   //    movement227ExecutabilityRight : Bool;   // Setup screen: executability of movement right
   //    movement228ExecutabilityLeft : Bool;   // Setup screen: executability of movement left
   //    movement228ExecutabilityRight : Bool;   // Setup screen: executability of movement right
   //    movement229ExecutabilityLeft : Bool;   // Setup screen: executability of movement left
   //    movement229ExecutabilityRight : Bool;   // Setup screen: executability of movement right
   //    movement230ExecutabilityLeft : Bool;   // Setup screen: executability of movement left
   //    movement230ExecutabilityRight : Bool;   // Setup screen: executability of movement right
   //    movement231ExecutabilityLeft : Bool;   // Setup screen: executability of movement left
   //    movement231ExecutabilityRight : Bool;   // Setup screen: executability of movement right
   //    movement232ExecutabilityLeft : Bool;   // Setup screen: executability of movement left
   //    movement232ExecutabilityRight : Bool;   // Setup screen: executability of movement right
   //    movement233ExecutabilityLeft : Bool;   // Setup screen: executability of movement left
   //    movement233ExecutabilityRight : Bool;   // Setup screen: executability of movement right
   //    movement234ExecutabilityLeft : Bool;   // Setup screen: executability of movement left
   //    movement234ExecutabilityRight : Bool;   // Setup screen: executability of movement right
   //    movement235ExecutabilityLeft : Bool;   // Setup screen: executability of movement left
   //    movement235ExecutabilityRight : Bool;   // Setup screen: executability of movement right
   //    movement236ExecutabilityLeft : Bool;   // Setup screen: executability of movement left
   //    movement236ExecutabilityRight : Bool;   // Setup screen: executability of movement right
   //    movement237ExecutabilityLeft : Bool;   // Setup screen: executability of movement left
   //    movement237ExecutabilityRight : Bool;   // Setup screen: executability of movement right
   //    movement238ExecutabilityLeft : Bool;   // Setup screen: executability of movement left
   //    movement238ExecutabilityRight : Bool;   // Setup screen: executability of movement right
   //    movement239ExecutabilityLeft : Bool;   // Setup screen: executability of movement left
   //    movement239ExecutabilityRight : Bool;   // Setup screen: executability of movement right
   //    movement240ExecutabilityLeft : Bool;   // Setup screen: executability of movement left
   //    movement240ExecutabilityRight : Bool;   // Setup screen: executability of movement right
   //    movement241ExecutabilityLeft : Bool;   // Setup screen: executability of movement left
   //    movement241ExecutabilityRight : Bool;   // Setup screen: executability of movement right
   //    movement242ExecutabilityLeft : Bool;   // Setup screen: executability of movement left
   //    movement242ExecutabilityRight : Bool;   // Setup screen: executability of movement right
   //    movement243ExecutabilityLeft : Bool;   // Setup screen: executability of movement left
   //    movement243ExecutabilityRight : Bool;   // Setup screen: executability of movement right
   //    movement244ExecutabilityLeft : Bool;   // Setup screen: executability of movement left
   //    movement244ExecutabilityRight : Bool;   // Setup screen: executability of movement right
   //    movement245ExecutabilityLeft : Bool;   // Setup screen: executability of movement left
   //    movement245ExecutabilityRight : Bool;   // Setup screen: executability of movement right
   //    movement246ExecutabilityLeft : Bool;   // Setup screen: executability of movement left
   //    movement246ExecutabilityRight : Bool;   // Setup screen: executability of movement right
   //    movement247ExecutabilityLeft : Bool;   // Setup screen: executability of movement left
   //    movement247ExecutabilityRight : Bool;   // Setup screen: executability of movement right
   //    movement248ExecutabilityLeft : Bool;   // Setup screen: executability of movement left
   //    movement248ExecutabilityRight : Bool;   // Setup screen: executability of movement right
   //    movement249ExecutabilityLeft : Bool;   // Setup screen: executability of movement left
   //    movement249ExecutabilityRight : Bool;   // Setup screen: executability of movement right
   //    movement250ExecutabilityLeft : Bool;   // Setup screen: executability of movement left
   //    movement250ExecutabilityRight : Bool;   // Setup screen: executability of movement right
   //    movement251ExecutabilityLeft : Bool;   // Setup screen: executability of movement left
   //    movement251ExecutabilityRight : Bool;   // Setup screen: executability of movement right
   //    movement252ExecutabilityLeft : Bool;   // Setup screen: executability of movement left
   //    movement252ExecutabilityRight : Bool;   // Setup screen: executability of movement right
   //    movement253ExecutabilityLeft : Bool;   // Setup screen: executability of movement left
   //    movement253ExecutabilityRight : Bool;   // Setup screen: executability of movement right
   //    movement254ExecutabilityLeft : Bool;   // Setup screen: executability of movement left
   //    movement254ExecutabilityRight : Bool;   // Setup screen: executability of movement right
   //    movement255ExecutabilityLeft : Bool;   // Setup screen: executability of movement left
   //    movement255ExecutabilityRight : Bool;   // Setup screen: executability of movement right
   //    movement256ExecutabilityLeft : Bool;   // Setup screen: executability of movement left
   //    movement256ExecutabilityRight : Bool;   // Setup screen: executability of movement right
   //    res_21 : Array[262..297] of Byte;
   //    res298 : Word;
   //    res_300 : Array[300..365] of Byte;
   //    movement : Array[1..6] of Word;
   //    movementControl : Word;
   //    versionFC57_0 : Byte;
   //    versionFC57_1 : Byte;
   //    versionFB451_0 : Byte;
   //    versionFB451_1 : Byte;
   //    res396 : Array[384..429] of Byte;
   //    clampingStationVarLayout : Array[1..40] of Word;
   //    res510 : Word;
   //    clampingStationNotPresent1 : Bool;
   //    clampingStationNotOk1 : Bool;
   //    clampingStationNotPresent2 : Bool;
   //    clampingStationNotOk2 : Bool;
   //    clampingStationNotPresent3 : Bool;
   //    clampingStationNotOk3 : Bool;
   //    clampingStationNotPresent4 : Bool;
   //    clampingStationNotOk4 : Bool;
   //    clampingStationNotPresent5 : Bool;
   //    clampingStationNotOk5 : Bool;
   //    clampingStationNotPresent6 : Bool;
   //    clampingStationNotOk6 : Bool;
   //    clampingStationNotPresent7 : Bool;
   //    clampingStationNotOk7 : Bool;
   //    clampingStationNotPresent8 : Bool;
   //    clampingStationNotOk8 : Bool;
   //    clampingStationNotPresent9 : Bool;
   //    clampingStationNotOk9 : Bool;
   //    clampingStationNotPresent10 : Bool;
   //    clampingStationNotOk10 : Bool;
   //    clampingStationNotPresent11 : Bool;
   //    clampingStationNotOk11 : Bool;
   //    clampingStationNotPresent12 : Bool;
   //    clampingStationNotOk12 : Bool;
   //    clampingStationNotPresent13 : Bool;
   //    clampingStationNotOk13 : Bool;
   //    clampingStationNotPresent14 : Bool;
   //    clampingStationNotOk14 : Bool;
   //    clampingStationNotPresent15 : Bool;
   //    clampingStationNotOk15 : Bool;
   //    clampingStationNotPresent16 : Bool;
   //    clampingStationNotOk16 : Bool;
   //    clampingStationNotPresent17 : Bool;
   //    clampingStationNotOk17 : Bool;
   //    clampingStationNotPresent18 : Bool;
   //    clampingStationNotOk18 : Bool;
   //    clampingStationNotPresent19 : Bool;
   //    clampingStationNotOk19 : Bool;
   //    clampingStationNotPresent20 : Bool;
   //    clampingStationNotOk20 : Bool;
   //    clampingStationNotPresent21 : Bool;
   //    clampingStationNotOk21 : Bool;
   //    clampingStationNotPresent22 : Bool;
   //    clampingStationNotOk22 : Bool;
   //    clampingStationNotPresent23 : Bool;
   //    clampingStationNotOk23 : Bool;
   //    clampingStationNotPresent24 : Bool;
   //    clampingStationNotOk24 : Bool;
   //    clampingStationNotPresent25 : Bool;
   //    clampingStationNotOk25 : Bool;
   //    clampingStationNotPresent26 : Bool;
   //    clampingStationNotOk26 : Bool;
   //    clampingStationNotPresent27 : Bool;
   //    clampingStationNotOk27 : Bool;
   //    clampingStationNotPresent28 : Bool;
   //    clampingStationNotOk28 : Bool;
   //    clampingStationNotPresent29 : Bool;
   //    clampingStationNotOk29 : Bool;
   //    clampingStationNotPresent30 : Bool;
   //    clampingStationNotOk30 : Bool;
   //    clampingStationNotPresent31 : Bool;
   //    clampingStationNotOk31 : Bool;
   //    clampingStationNotPresent32 : Bool;
   //    clampingStationNotOk32 : Bool;
   //    clampingStationNotPresent33 : Bool;
   //    clampingStationNotOk33 : Bool;
   //    clampingStationNotPresent34 : Bool;
   //    clampingStationNotOk34 : Bool;
   //    clampingStationNotPresent35 : Bool;
   //    clampingStationNotOk35 : Bool;
   //    clampingStationNotPresent36 : Bool;
   //    clampingStationNotOk36 : Bool;
   //    clampingStationNotPresent37 : Bool;
   //    clampingStationNotOk37 : Bool;
   //    clampingStationNotPresent38 : Bool;
   //    clampingStationNotOk38 : Bool;
   //    clampingStationNotPresent39 : Bool;
   //    clampingStationNotOk39 : Bool;
   //    clampingStationNotPresent40 : Bool;
   //    clampingStationNotOk40 : Bool;
   //    rs_522 : Bool;
   //    rs_5221 : Bool;
   //    rs_5222 : Bool;
   //    rs_5223 : Bool;
   //    rs_5224 : Bool;
   //    rs_5225 : Bool;
   //    rs_5226 : Bool;
   //    rs_5227 : Bool;
   //    movement1ActiveLeft : Bool;   // Movement left active
   //    movement1ActiveRight : Bool;   // Movement right active
   //    movement2ActiveLeft : Bool;   // Movement left active
   //    movement2ActiveRight : Bool;   // Movement right active
   //    movement3ActiveLeft : Bool;   // Movement left active
   //    movement3ActiveRight : Bool;   // Movement right active
   //    movement4ActiveLeft : Bool;   // Movement left active
   //    movement4ActiveRight : Bool;   // Movement right active
   //    movement5ActiveLeft : Bool;   // Movement left active
   //    movement5ActiveRight : Bool;   // Movement right active
   //    movement6ActiveLeft : Bool;   // Movement left active
   //    movement6ActiveRight : Bool;   // Movement right active
   //    movement7ActiveLeft : Bool;   // Movement left active
   //    movement7ActiveRight : Bool;   // Movement right active
   //    movement8ActiveLeft : Bool;   // Movement left active
   //    movement8ActiveRight : Bool;   // Movement right active
   //    movement9ActiveLeft : Bool;   // Movement left active
   //    movement9ActiveRight : Bool;   // Movement right active
   //    movement10ActiveLeft : Bool;   // Movement left active
   //    movement10ActiveRight : Bool;   // Movement right active
   //    movement11ActiveLeft : Bool;   // Movement left active
   //    movement11ActiveRight : Bool;   // Movement right active
   //    movement12ActiveLeft : Bool;   // Movement left active
   //    movement12ActiveRight : Bool;   // Movement right active
   //    movement13ActiveLeft : Bool;   // Movement left active
   //    movement13ActiveRight : Bool;   // Movement right active
   //    movement14ActiveLeft : Bool;   // Movement left active
   //    movement14ActiveRight : Bool;   // Movement right active
   //    movement15ActiveLeft : Bool;   // Movement left active
   //    movement15ActiveRight : Bool;   // Movement right active
   //    movement16ActiveLeft : Bool;   // Movement left active
   //    movement16ActiveRight : Bool;   // Movement right active
   //    movement17ActiveLeft : Bool;   // Movement left active
   //    movement17ActiveRight : Bool;   // Movement right active
   //    movement18ActiveLeft : Bool;   // Movement left active
   //    movement18ActiveRight : Bool;   // Movement right active
   //    movement19ActiveLeft : Bool;   // Movement left active
   //    movement19ActiveRight : Bool;   // Movement right active
   //    movement20ActiveLeft : Bool;   // Movement left active
   //    movement20ActiveRight : Bool;   // Movement right active
   //    movement21ActiveLeft : Bool;   // Movement left active
   //    movement21ActiveRight : Bool;   // Movement right active
   //    movement22ActiveLeft : Bool;   // Movement left active
   //    movement22ActiveRight : Bool;   // Movement right active
   //    movement23ActiveLeft : Bool;   // Movement left active
   //    movement23ActiveRight : Bool;   // Movement right active
   //    movement24ActiveLeft : Bool;   // Movement left active
   //    movement24ActiveRight : Bool;   // Movement right active
   //    movement25ActiveLeft : Bool;   // Movement left active
   //    movement25ActiveRight : Bool;   // Movement right active
   //    movement26ActiveLeft : Bool;   // Movement left active
   //    movement26ActiveRight : Bool;   // Movement right active
   //    movement27ActiveLeft : Bool;   // Movement left active
   //    movement27ActiveRight : Bool;   // Movement right active
   //    movement28ActiveLeft : Bool;   // Movement left active
   //    movement28ActiveRight : Bool;   // Movement right active
   //    movement29ActiveLeft : Bool;   // Movement left active
   //    movement29ActiveRight : Bool;   // Movement right active
   //    movement30ActiveLeft : Bool;   // Movement left active
   //    movement30ActiveRight : Bool;   // Movement right active
   //    movement31ActiveLeft : Bool;   // Movement left active
   //    movement31ActiveRight : Bool;   // Movement right active
   //    movement32ActiveLeft : Bool;   // Movement left active
   //    movement32ActiveRight : Bool;   // Movement right active
   //    movement33ActiveLeft : Bool;   // Movement left active
   //    movement33ActiveRight : Bool;   // Movement right active
   //    movement34ActiveLeft : Bool;   // Movement left active
   //    movement34ActiveRight : Bool;   // Movement right active
   //    movement35ActiveLeft : Bool;   // Movement left active
   //    movement35ActiveRight : Bool;   // Movement right active
   //    movement36ActiveLeft : Bool;   // Movement left active
   //    movement36ActiveRight : Bool;   // Movement right active
   //    movement37ActiveLeft : Bool;   // Movement left active
   //    movement37ActiveRight : Bool;   // Movement right active
   //    movement38ActiveLeft : Bool;   // Movement left active
   //    movement38ActiveRight : Bool;   // Movement right active
   //    movement39ActiveLeft : Bool;   // Movement left active
   //    movement39ActiveRight : Bool;   // Movement right active
   //    movement40ActiveLeft : Bool;   // Movement left active
   //    movement40ActiveRight : Bool;   // Movement right active
   //    movement41ActiveLeft : Bool;   // Movement left active
   //    movement41ActiveRight : Bool;   // Movement right active
   //    movement42ActiveLeft : Bool;   // Movement left active
   //    movement42ActiveRight : Bool;   // Movement right active
   //    movement43ActiveLeft : Bool;   // Movement left active
   //    movement43ActiveRight : Bool;   // Movement right active
   //    movement44ActiveLeft : Bool;   // Movement left active
   //    movement44ActiveRight : Bool;   // Movement right active
   //    movement45ActiveLeft : Bool;   // Movement left active
   //    movement45ActiveRight : Bool;   // Movement right active
   //    movement46ActiveLeft : Bool;   // Movement left active
   //    movement46ActiveRight : Bool;   // Movement right active
   //    movement47ActiveLeft : Bool;   // Movement left active
   //    movement47ActiveRight : Bool;   // Movement right active
   //    movement48ActiveLeft : Bool;   // Movement left active
   //    movement48ActiveRight : Bool;   // Movement right active
   //    movement49ActiveLeft : Bool;   // Movement left active
   //    movement49ActiveRight : Bool;   // Movement right active
   //    movement50ActiveLeft : Bool;   // Movement left active
   //    movement50ActiveRight : Bool;   // Movement right active
   //    movement51ActiveLeft : Bool;   // Movement left active
   //    movement51ActiveRight : Bool;   // Movement right active
   //    movement52ActiveLeft : Bool;   // Movement left active
   //    movement52ActiveRight : Bool;   // Movement right active
   //    movement53ActiveLeft : Bool;   // Movement left active
   //    movement53ActiveRight : Bool;   // Movement right active
   //    movement54ActiveLeft : Bool;   // Movement left active
   //    movement54ActiveRight : Bool;   // Movement right active
   //    movement55ActiveLeft : Bool;   // Movement left active
   //    movement55ActiveRight : Bool;   // Movement right active
   //    movement56ActiveLeft : Bool;   // Movement left active
   //    movement56ActiveRight : Bool;   // Movement right active
   //    movement57ActiveLeft : Bool;   // Movement left active
   //    movement57ActiveRight : Bool;   // Movement right active
   //    movement58ActiveLeft : Bool;   // Movement left active
   //    movement58ActiveRight : Bool;   // Movement right active
   //    movement59ActiveLeft : Bool;   // Movement left active
   //    movement59ActiveRight : Bool;   // Movement right active
   //    movement60ActiveLeft : Bool;   // Movement left active
   //    movement60ActiveRight : Bool;   // Movement right active
   //    movement61ActiveLeft : Bool;   // Movement left active
   //    movement61ActiveRight : Bool;   // Movement right active
   //    movement62ActiveLeft : Bool;   // Movement left active
   //    movement62ActiveRight : Bool;   // Movement right active
   //    movement63ActiveLeft : Bool;   // Movement left active
   //    movement63ActiveRight : Bool;   // Movement right active
   //    movement64ActiveLeft : Bool;   // Movement left active
   //    movement64ActiveRight : Bool;   // Movement right active
   //    movement65ActiveLeft : Bool;   // Movement left active
   //    movement65ActiveRight : Bool;   // Movement right active
   //    movement66ActiveLeft : Bool;   // Movement left active
   //    movement66ActiveRight : Bool;   // Movement right active
   //    movement67ActiveLeft : Bool;   // Movement left active
   //    movement67ActiveRight : Bool;   // Movement right active
   //    movement68ActiveLeft : Bool;   // Movement left active
   //    movement68ActiveRight : Bool;   // Movement right active
   //    movement69ActiveLeft : Bool;   // Movement left active
   //    movement69ActiveRight : Bool;   // Movement right active
   //    movement70ActiveLeft : Bool;   // Movement left active
   //    movement70ActiveRight : Bool;   // Movement right active
   //    movement71ActiveLeft : Bool;   // Movement left active
   //    movement71ActiveRight : Bool;   // Movement right active
   //    movement72ActiveLeft : Bool;   // Movement left active
   //    movement72ActiveRight : Bool;   // Movement right active
   //    movement73ActiveLeft : Bool;   // Movement left active
   //    movement73ActiveRight : Bool;   // Movement right active
   //    movement74ActiveLeft : Bool;   // Movement left active
   //    movement74ActiveRight : Bool;   // Movement right active
   //    movement75ActiveLeft : Bool;   // Movement left active
   //    movement75ActiveRight : Bool;   // Movement right active
   //    movement76ActiveLeft : Bool;   // Movement left active
   //    movement76ActiveRight : Bool;   // Movement right active
   //    movement77ActiveLeft : Bool;   // Movement left active
   //    movement77ActiveRight : Bool;   // Movement right active
   //    movement78ActiveLeft : Bool;   // Movement left active
   //    movement78ActiveRight : Bool;   // Movement right active
   //    movement79ActiveLeft : Bool;   // Movement left active
   //    movement79ActiveRight : Bool;   // Movement right active
   //    movement80ActiveLeft : Bool;   // Movement left active
   //    movement80ActiveRight : Bool;   // Movement right active
   //    movement81ActiveLeft : Bool;   // Movement left active
   //    movement81ActiveRight : Bool;   // Movement right active
   //    movement82ActiveLeft : Bool;   // Movement left active
   //    movement82ActiveRight : Bool;   // Movement right active
   //    movement83ActiveLeft : Bool;   // Movement left active
   //    movement83ActiveRight : Bool;   // Movement right active
   //    movement84ActiveLeft : Bool;   // Movement left active
   //    movement84ActiveRight : Bool;   // Movement right active
   //    movement85ActiveLeft : Bool;   // Movement left active
   //    movement85ActiveRight : Bool;   // Movement right active
   //    movement86ActiveLeft : Bool;   // Movement left active
   //    movement86ActiveRight : Bool;   // Movement right active
   //    movement87ActiveLeft : Bool;   // Movement left active
   //    movement87ActiveRight : Bool;   // Movement right active
   //    movement88ActiveLeft : Bool;   // Movement left active
   //    movement88ActiveRight : Bool;   // Movement right active
   //    movement89ActiveLeft : Bool;   // Movement left active
   //    movement89ActiveRight : Bool;   // Movement right active
   //    movement90ActiveLeft : Bool;   // Movement left active
   //    movement90ActiveRight : Bool;   // Movement right active
   //    movement91ActiveLeft : Bool;   // Movement left active
   //    movement91ActiveRight : Bool;   // Movement right active
   //    movement92ActiveLeft : Bool;   // Movement left active
   //    movement92ActiveRight : Bool;   // Movement right active
   //    movement93ActiveLeft : Bool;   // Movement left active
   //    movement93ActiveRight : Bool;   // Movement right active
   //    movement94ActiveLeft : Bool;   // Movement left active
   //    movement94ActiveRight : Bool;   // Movement right active
   //    movement95ActiveLeft : Bool;   // Movement left active
   //    movement95ActiveRight : Bool;   // Movement right active
   //    movement96ActiveLeft : Bool;   // Movement left active
   //    movement96ActiveRight : Bool;   // Movement right active
   //    movement97ActiveLeft : Bool;   // Movement left active
   //    movement97ActiveRight : Bool;   // Movement right active
   //    movement98ActiveLeft : Bool;   // Movement left active
   //    movement98ActiveRight : Bool;   // Movement right active
   //    movement99ActiveLeft : Bool;   // Movement left active
   //    movement99ActiveRight : Bool;   // Movement right active
   //    movement100ActiveLeft : Bool;   // Movement left active
   //    movement100ActiveRight : Bool;   // Movement right active
   //    movement101ActiveLeft : Bool;   // Movement left active
   //    movement101ActiveRight : Bool;   // Movement right active
   //    movement102ActiveLeft : Bool;   // Movement left active
   //    movement102ActiveRight : Bool;   // Movement right active
   //    movement103ActiveLeft : Bool;   // Movement left active
   //    movement103ActiveRight : Bool;   // Movement right active
   //    movement104ActiveLeft : Bool;   // Movement left active
   //    movement104ActiveRight : Bool;   // Movement right active
   //    movement105ActiveLeft : Bool;   // Movement left active
   //    movement105ActiveRight : Bool;   // Movement right active
   //    movement106ActiveLeft : Bool;   // Movement left active
   //    movement106ActiveRight : Bool;   // Movement right active
   //    movement107ActiveLeft : Bool;   // Movement left active
   //    movement107ActiveRight : Bool;   // Movement right active
   //    movement108ActiveLeft : Bool;   // Movement left active
   //    movement108ActiveRight : Bool;   // Movement right active
   //    movement109ActiveLeft : Bool;   // Movement left active
   //    movement109ActiveRight : Bool;   // Movement right active
   //    movement110ActiveLeft : Bool;   // Movement left active
   //    movement110ActiveRight : Bool;   // Movement right active
   //    movement111ActiveLeft : Bool;   // Movement left active
   //    movement111ActiveRight : Bool;   // Movement right active
   //    movement112ActiveLeft : Bool;   // Movement left active
   //    movement112ActiveRight : Bool;   // Movement right active
   //    movement113ActiveLeft : Bool;   // Movement left active
   //    movement113ActiveRight : Bool;   // Movement right active
   //    movement114ActiveLeft : Bool;   // Movement left active
   //    movement114ActiveRight : Bool;   // Movement right active
   //    movement115ActiveLeft : Bool;   // Movement left active
   //    movement115ActiveRight : Bool;   // Movement right active
   //    movement116ActiveLeft : Bool;   // Movement left active
   //    movement116ActiveRight : Bool;   // Movement right active
   //    movement117ActiveLeft : Bool;   // Movement left active
   //    movement117ActiveRight : Bool;   // Movement right active
   //    movement118ActiveLeft : Bool;   // Movement left active
   //    movement118ActiveRight : Bool;   // Movement right active
   //    movement119ActiveLeft : Bool;   // Movement left active
   //    movement119ActiveRight : Bool;   // Movement right active
   //    movement120ActiveLeft : Bool;   // Movement left active
   //    movement120ActiveRight : Bool;   // Movement right active
   //    movement121ActiveLeft : Bool;   // Movement left active
   //    movement121ActiveRight : Bool;   // Movement right active
   //    movement122ActiveLeft : Bool;   // Movement left active
   //    movement122ActiveRight : Bool;   // Movement right active
   //    movement123ActiveLeft : Bool;   // Movement left active
   //    movement123ActiveRight : Bool;   // Movement right active
   //    movement124ActiveLeft : Bool;   // Movement left active
   //    movement124ActiveRight : Bool;   // Movement right active
   //    movement125ActiveLeft : Bool;   // Movement left active
   //    movement125ActiveRight : Bool;   // Movement right active
   //    movement126ActiveLeft : Bool;   // Movement left active
   //    movement126ActiveRight : Bool;   // Movement right active
   //    movement127ActiveLeft : Bool;   // Movement left active
   //    movement127ActiveRight : Bool;   // Movement right active
   //    movement128ActiveLeft : Bool;   // Movement left active
   //    movement128ActiveRight : Bool;   // Movement right active
   //    movement129ActiveLeft : Bool;   // Movement left active
   //    movement129ActiveRight : Bool;   // Movement right active
   //    movement130ActiveLeft : Bool;   // Movement left active
   //    movement130ActiveRight : Bool;   // Movement right active
   //    movement131ActiveLeft : Bool;   // Movement left active
   //    movement131ActiveRight : Bool;   // Movement right active
   //    movement132ActiveLeft : Bool;   // Movement left active
   //    movement132ActiveRight : Bool;   // Movement right active
   //    movement133ActiveLeft : Bool;   // Movement left active
   //    movement133ActiveRight : Bool;   // Movement right active
   //    movement134ActiveLeft : Bool;   // Movement left active
   //    movement134ActiveRight : Bool;   // Movement right active
   //    movement135ActiveLeft : Bool;   // Movement left active
   //    movement135ActiveRight : Bool;   // Movement right active
   //    movement136ActiveLeft : Bool;   // Movement left active
   //    movement136ActiveRight : Bool;   // Movement right active
   //    movement137ActiveLeft : Bool;   // Movement left active
   //    movement137ActiveRight : Bool;   // Movement right active
   //    movement138ActiveLeft : Bool;   // Movement left active
   //    movement138ActiveRight : Bool;   // Movement right active
   //    movement139ActiveLeft : Bool;   // Movement left active
   //    movement139ActiveRight : Bool;   // Movement right active
   //    movement140ActiveLeft : Bool;   // Movement left active
   //    movement140ActiveRight : Bool;   // Movement right active
   //    movement141ActiveLeft : Bool;   // Movement left active
   //    movement141ActiveRight : Bool;   // Movement right active
   //    movement142ActiveLeft : Bool;   // Movement left active
   //    movement142ActiveRight : Bool;   // Movement right active
   //    movement143ActiveLeft : Bool;   // Movement left active
   //    movement143ActiveRight : Bool;   // Movement right active
   //    movement144ActiveLeft : Bool;   // Movement left active
   //    movement144ActiveRight : Bool;   // Movement right active
   //    movement145ActiveLeft : Bool;   // Movement left active
   //    movement145ActiveRight : Bool;   // Movement right active
   //    movement146ActiveLeft : Bool;   // Movement left active
   //    movement146ActiveRight : Bool;   // Movement right active
   //    movement147ActiveLeft : Bool;   // Movement left active
   //    movement147ActiveRight : Bool;   // Movement right active
   //    movement148ActiveLeft : Bool;   // Movement left active
   //    movement148ActiveRight : Bool;   // Movement right active
   //    movement149ActiveLeft : Bool;   // Movement left active
   //    movement149ActiveRight : Bool;   // Movement right active
   //    movement150ActiveLeft : Bool;   // Movement left active
   //    movement150ActiveRight : Bool;   // Movement right active
   //    movement151ActiveLeft : Bool;   // Movement left active
   //    movement151ActiveRight : Bool;   // Movement right active
   //    movement152ActiveLeft : Bool;   // Movement left active
   //    movement152ActiveRight : Bool;   // Movement right active
   //    movement153ActiveLeft : Bool;   // Movement left active
   //    movement153ActiveRight : Bool;   // Movement right active
   //    movement154ActiveLeft : Bool;   // Movement left active
   //    movement154ActiveRight : Bool;   // Movement right active
   //    movement155ActiveLeft : Bool;   // Movement left active
   //    movement155ActiveRight : Bool;   // Movement right active
   //    movement156ActiveLeft : Bool;   // Movement left active
   //    movement156ActiveRight : Bool;   // Movement right active
   //    movement157ActiveLeft : Bool;   // Movement left active
   //    movement157ActiveRight : Bool;   // Movement right active
   //    movement158ActiveLeft : Bool;   // Movement left active
   //    movement158ActiveRight : Bool;   // Movement right active
   //    movement159ActiveLeft : Bool;   // Movement left active
   //    movement159ActiveRight : Bool;   // Movement right active
   //    movement160ActiveLeft : Bool;   // Movement left active
   //    movement160ActiveRight : Bool;   // Movement right active
   //    movement161ActiveLeft : Bool;   // Movement left active
   //    movement161ActiveRight : Bool;   // Movement right active
   //    movement162ActiveLeft : Bool;   // Movement left active
   //    movement162ActiveRight : Bool;   // Movement right active
   //    movement163ActiveLeft : Bool;   // Movement left active
   //    movement163ActiveRight : Bool;   // Movement right active
   //    movement164ActiveLeft : Bool;   // Movement left active
   //    movement164ActiveRight : Bool;   // Movement right active
   //    movement165ActiveLeft : Bool;   // Movement left active
   //    movement165ActiveRight : Bool;   // Movement right active
   //    movement166ActiveLeft : Bool;   // Movement left active
   //    movement166ActiveRight : Bool;   // Movement right active
   //    movement167ActiveLeft : Bool;   // Movement left active
   //    movement167ActiveRight : Bool;   // Movement right active
   //    movement168ActiveLeft : Bool;   // Movement left active
   //    movement168ActiveRight : Bool;   // Movement right active
   //    movement169ActiveLeft : Bool;   // Movement left active
   //    movement169ActiveRight : Bool;   // Movement right active
   //    movement170ActiveLeft : Bool;   // Movement left active
   //    movement170ActiveRight : Bool;   // Movement right active
   //    movement171ActiveLeft : Bool;   // Movement left active
   //    movement171ActiveRight : Bool;   // Movement right active
   //    movement172ActiveLeft : Bool;   // Movement left active
   //    movement172ActiveRight : Bool;   // Movement right active
   //    movement173ActiveLeft : Bool;   // Movement left active
   //    movement173ActiveRight : Bool;   // Movement right active
   //    movement174ActiveLeft : Bool;   // Movement left active
   //    movement174ActiveRight : Bool;   // Movement right active
   //    movement175ActiveLeft : Bool;   // Movement left active
   //    movement175ActiveRight : Bool;   // Movement right active
   //    movement176ActiveLeft : Bool;   // Movement left active
   //    movement176ActiveRight : Bool;   // Movement right active
   //    movement177ActiveLeft : Bool;   // Movement left active
   //    movement177ActiveRight : Bool;   // Movement right active
   //    movement178ActiveLeft : Bool;   // Movement left active
   //    movement178ActiveRight : Bool;   // Movement right active
   //    movement179ActiveLeft : Bool;   // Movement left active
   //    movement179ActiveRight : Bool;   // Movement right active
   //    movement180ActiveLeft : Bool;   // Movement left active
   //    movement180ActiveRight : Bool;   // Movement right active
   //    movement181ActiveLeft : Bool;   // Movement left active
   //    movement181ActiveRight : Bool;   // Movement right active
   //    movement182ActiveLeft : Bool;   // Movement left active
   //    movement182ActiveRight : Bool;   // Movement right active
   //    movement183ActiveLeft : Bool;   // Movement left active
   //    movement183ActiveRight : Bool;   // Movement right active
   //    movement184ActiveLeft : Bool;   // Movement left active
   //    movement184ActiveRight : Bool;   // Movement right active
   //    movement185ActiveLeft : Bool;   // Movement left active
   //    movement185ActiveRight : Bool;   // Movement right active
   //    movement186ActiveLeft : Bool;   // Movement left active
   //    movement186ActiveRight : Bool;   // Movement right active
   //    movement187ActiveLeft : Bool;   // Movement left active
   //    movement187ActiveRight : Bool;   // Movement right active
   //    movement188ActiveLeft : Bool;   // Movement left active
   //    movement188ActiveRight : Bool;   // Movement right active
   //    movement189ActiveLeft : Bool;   // Movement left active
   //    movement189ActiveRight : Bool;   // Movement right active
   //    movement190ActiveLeft : Bool;   // Movement left active
   //    movement190ActiveRight : Bool;   // Movement right active
   //    movement191ActiveLeft : Bool;   // Movement left active
   //    movement191ActiveRight : Bool;   // Movement right active
   //    movement192ActiveLeft : Bool;   // Movement left active
   //    movement192ActiveRight : Bool;   // Movement right active
   //    movement193ActiveLeft : Bool;   // Movement left active
   //    movement193ActiveRight : Bool;   // Movement right active
   //    movement194ActiveLeft : Bool;   // Movement left active
   //    movement194ActiveRight : Bool;   // Movement right active
   //    movement195ActiveLeft : Bool;   // Movement left active
   //    movement195ActiveRight : Bool;   // Movement right active
   //    movement196ActiveLeft : Bool;   // Movement left active
   //    movement196ActiveRight : Bool;   // Movement right active
   //    movement197ActiveLeft : Bool;   // Movement left active
   //    movement197ActiveRight : Bool;   // Movement right active
   //    movement198ActiveLeft : Bool;   // Movement left active
   //    movement198ActiveRight : Bool;   // Movement right active
   //    movement199ActiveLeft : Bool;   // Movement left active
   //    movement199ActiveRight : Bool;   // Movement right active
   //    movement200ActiveLeft : Bool;   // Movement left active
   //    movement200ActiveRight : Bool;   // Movement right active
   //    movement201ActiveLeft : Bool;   // Movement left active
   //    movement201ActiveRight : Bool;   // Movement right active
   //    movement202ActiveLeft : Bool;   // Movement left active
   //    movement202ActiveRight : Bool;   // Movement right active
   //    movement203ActiveLeft : Bool;   // Movement left active
   //    movement203ActiveRight : Bool;   // Movement right active
   //    movement204ActiveLeft : Bool;   // Movement left active
   //    movement204ActiveRight : Bool;   // Movement right active
   //    movement205ActiveLeft : Bool;   // Movement left active
   //    movement205ActiveRight : Bool;   // Movement right active
   //    movement206ActiveLeft : Bool;   // Movement left active
   //    movement206ActiveRight : Bool;   // Movement right active
   //    movement207ActiveLeft : Bool;   // Movement left active
   //    movement207ActiveRight : Bool;   // Movement right active
   //    movement208ActiveLeft : Bool;   // Movement left active
   //    movement208ActiveRight : Bool;   // Movement right active
   //    movement209ActiveLeft : Bool;   // Movement left active
   //    movement209ActiveRight : Bool;   // Movement right active
   //    movement210ActiveLeft : Bool;   // Movement left active
   //    movement210ActiveRight : Bool;   // Movement right active
   //    movement211ActiveLeft : Bool;   // Movement left active
   //    movement211ActiveRight : Bool;   // Movement right active
   //    movement212ActiveLeft : Bool;   // Movement left active
   //    movement212ActiveRight : Bool;   // Movement right active
   //    movement213ActiveLeft : Bool;   // Movement left active
   //    movement213ActiveRight : Bool;   // Movement right active
   //    movement214ActiveLeft : Bool;   // Movement left active
   //    movement214ActiveRight : Bool;   // Movement right active
   //    movement215ActiveLeft : Bool;   // Movement left active
   //    movement215ActiveRight : Bool;   // Movement right active
   //    movement216ActiveLeft : Bool;   // Movement left active
   //    movement216ActiveRight : Bool;   // Movement right active
   //    movement217ActiveLeft : Bool;   // Movement left active
   //    movement217ActiveRight : Bool;   // Movement right active
   //    movement218ActiveLeft : Bool;   // Movement left active
   //    movement218ActiveRight : Bool;   // Movement right active
   //    movement219ActiveLeft : Bool;   // Movement left active
   //    movement219ActiveRight : Bool;   // Movement right active
   //    movement220ActiveLeft : Bool;   // Movement left active
   //    movement220ActiveRight : Bool;   // Movement right active
   //    movement221ActiveLeft : Bool;   // Movement left active
   //    movement221ActiveRight : Bool;   // Movement right active
   //    movement222ActiveLeft : Bool;   // Movement left active
   //    movement222ActiveRight : Bool;   // Movement right active
   //    movement223ActiveLeft : Bool;   // Movement left active
   //    movement223ActiveRight : Bool;   // Movement right active
   //    movement224ActiveLeft : Bool;   // Movement left active
   //    movement224ActiveRight : Bool;   // Movement right active
   //    movement225ActiveLeft : Bool;   // Movement left active
   //    movement225ActiveRight : Bool;   // Movement right active
   //    movement226ActiveLeft : Bool;   // Movement left active
   //    movement226ActiveRight : Bool;   // Movement right active
   //    movement227ActiveLeft : Bool;   // Movement left active
   //    movement227ActiveRight : Bool;   // Movement right active
   //    movement228ActiveLeft : Bool;   // Movement left active
   //    movement228ActiveRight : Bool;   // Movement right active
   //    movement229ActiveLeft : Bool;   // Movement left active
   //    movement229ActiveRight : Bool;   // Movement right active
   //    movement230ActiveLeft : Bool;   // Movement left active
   //    movement230ActiveRight : Bool;   // Movement right active
   //    movement231ActiveLeft : Bool;   // Movement left active
   //    movement231ActiveRight : Bool;   // Movement right active
   //    movement232ActiveLeft : Bool;   // Movement left active
   //    movement232ActiveRight : Bool;   // Movement right active
   //    movement233ActiveLeft : Bool;   // Movement left active
   //    movement233ActiveRight : Bool;   // Movement right active
   //    movement234ActiveLeft : Bool;   // Movement left active
   //    movement234ActiveRight : Bool;   // Movement right active
   //    movement235ActiveLeft : Bool;   // Movement left active
   //    movement235ActiveRight : Bool;   // Movement right active
   //    movement236ActiveLeft : Bool;   // Movement left active
   //    movement236ActiveRight : Bool;   // Movement right active
   //    movement237ActiveLeft : Bool;   // Movement left active
   //    movement237ActiveRight : Bool;   // Movement right active
   //    movement238ActiveLeft : Bool;   // Movement left active
   //    movement238ActiveRight : Bool;   // Movement right active
   //    movement239ActiveLeft : Bool;   // Movement left active
   //    movement239ActiveRight : Bool;   // Movement right active
   //    movement240ActiveLeft : Bool;   // Movement left active
   //    movement240ActiveRight : Bool;   // Movement right active
   //    movement241ActiveLeft : Bool;   // Movement left active
   //    movement241ActiveRight : Bool;   // Movement right active
   //    movement242ActiveLeft : Bool;   // Movement left active
   //    movement242ActiveRight : Bool;   // Movement right active
   //    movement243ActiveLeft : Bool;   // Movement left active
   //    movement243ActiveRight : Bool;   // Movement right active
   //    movement244ActiveLeft : Bool;   // Movement left active
   //    movement244ActiveRight : Bool;   // Movement right active
   //    movement245ActiveLeft : Bool;   // Movement left active
   //    movement245ActiveRight : Bool;   // Movement right active
   //    movement246ActiveLeft : Bool;   // Movement left active
   //    movement246ActiveRight : Bool;   // Movement right active
   //    movement247ActiveLeft : Bool;   // Movement left active
   //    movement247ActiveRight : Bool;   // Movement right active
   //    movement248ActiveLeft : Bool;   // Movement left active
   //    movement248ActiveRight : Bool;   // Movement right active
   //    movement249ActiveLeft : Bool;   // Movement left active
   //    movement249ActiveRight : Bool;   // Movement right active
   //    movement250ActiveLeft : Bool;   // Movement left active
   //    movement250ActiveRight : Bool;   // Movement right active
   //    movement251ActiveLeft : Bool;   // Movement left active
   //    movement251ActiveRight : Bool;   // Movement right active
   //    movement252ActiveLeft : Bool;   // Movement left active
   //    movement252ActiveRight : Bool;   // Movement right active
   //    movement253ActiveLeft : Bool;   // Movement left active
   //    movement253ActiveRight : Bool;   // Movement right active
   //    movement254ActiveLeft : Bool;   // Movement left active
   //    movement254ActiveRight : Bool;   // Movement right active
   //    movement255ActiveLeft : Bool;   // Movement left active
   //    movement255ActiveRight : Bool;   // Movement right active
   //    movement256ActiveLeft : Bool;   // Movement left active
   //    movement256ActiveRight : Bool;   // Movement right active
   //    nutRunnerGradientHigh1 : Bool;
   //    nutRunnerGradientLow1 : Bool;
   //    nutRunnerGradientHigh2 : Bool;
   //    nutRunnerGradientLow2 : Bool;
   //    nutRunnerGradientHigh3 : Bool;
   //    nutRunnerGradientLow3 : Bool;
   //    nutRunnerGradientHigh4 : Bool;
   //    nutRunnerGradientLow4 : Bool;
   //    nutRunnerGradientHigh5 : Bool;
   //    nutRunnerGradientLow5 : Bool;
   //    nutRunnerGradientHigh6 : Bool;
   //    nutRunnerGradientLow6 : Bool;
   //    nutRunnerGradientHigh7 : Bool;
   //    nutRunnerGradientLow7 : Bool;
   //    nutRunnerGradientHigh8 : Bool;
   //    nutRunnerGradientLow8 : Bool;
   //    nutRunnerGradientHigh9 : Bool;
   //    nutRunnerGradientLow9 : Bool;
   //    nutRunnerGradientHigh10 : Bool;
   //    nutRunnerGradientLow10 : Bool;
   //    nutRunnerGradientHigh11 : Bool;
   //    nutRunnerGradientLow11 : Bool;
   //    nutRunnerGradientHigh12 : Bool;
   //    nutRunnerGradientLow12 : Bool;
   //    nutRunnerGradientHigh13 : Bool;
   //    nutRunnerGradientLow13 : Bool;
   //    nutRunnerGradientHigh14 : Bool;
   //    nutRunnerGradientLow14 : Bool;
   //    nutRunnerGradientHigh15 : Bool;
   //    nutRunnerGradientLow15 : Bool;
   //    nutRunnerGradientHigh16 : Bool;
   //    nutRunnerGradientLow16 : Bool;
   //    nutRunnerGradientHigh17 : Bool;
   //    nutRunnerGradientLow17 : Bool;
   //    nutRunnerGradientHigh18 : Bool;
   //    nutRunnerGradientLow18 : Bool;
   //    nutRunnerGradientHigh19 : Bool;
   //    nutRunnerGradientLow19 : Bool;
   //    nutRunnerGradientHigh20 : Bool;
   //    nutRunnerGradientLow20 : Bool;
   //    nutRunnerGradientHigh21 : Bool;
   //    nutRunnerGradientLow21 : Bool;
   //    nutRunnerGradientHigh22 : Bool;
   //    nutRunnerGradientLow22 : Bool;
   //    nutRunnerGradientHigh23 : Bool;
   //    nutRunnerGradientLow23 : Bool;
   //    nutRunnerGradientHigh24 : Bool;
   //    nutRunnerGradientLow24 : Bool;
   //    nutRunnerGradientHigh25 : Bool;
   //    nutRunnerGradientLow25 : Bool;
   //    nutRunnerGradientHigh26 : Bool;
   //    nutRunnerGradientLow26 : Bool;
   //    nutRunnerGradientHigh27 : Bool;
   //    nutRunnerGradientLow27 : Bool;
   //    nutRunnerGradientHigh28 : Bool;
   //    nutRunnerGradientLow28 : Bool;
   //    nutRunnerGradientHigh29 : Bool;
   //    nutRunnerGradientLow29 : Bool;
   //    nutRunnerGradientHigh30 : Bool;
   //    nutRunnerGradientLow30 : Bool;
   //    nutRunnerGradientHigh31 : Bool;
   //    nutRunnerGradientLow31 : Bool;
   //    nutRunnerGradientHigh32 : Bool;
   //    nutRunnerGradientLow32 : Bool;
   //    nutRunnerGradientHigh33 : Bool;
   //    nutRunnerGradientLow33 : Bool;
   //    nutRunnerGradientHigh34 : Bool;
   //    nutRunnerGradientLow34 : Bool;
   //    nutRunnerGradientHigh35 : Bool;
   //    nutRunnerGradientLow35 : Bool;
   //    nutRunnerGradientHigh36 : Bool;
   //    nutRunnerGradientLow36 : Bool;
   //    nutRunnerGradientHigh37 : Bool;
   //    nutRunnerGradientLow37 : Bool;
   //    nutRunnerGradientHigh38 : Bool;
   //    nutRunnerGradientLow38 : Bool;
   //    nutRunnerGradientHigh39 : Bool;
   //    nutRunnerGradientLow39 : Bool;
   //    nutRunnerGradientHigh40 : Bool;
   //    nutRunnerGradientLow40 : Bool;
   //    res_598 : Array[598..605] of Byte;
   //    res_606 : Array[606..611] of Byte;
   //    res612 : Array[612..631] of Byte;
   //    res632 : Byte;
   //    comBitSettingTableHmiPlc : Bool;
   //    comBitTablePlcHmi : Bool;
   //    res_6332 : Bool;
   //    res_6333 : Bool;
   //    res_6334 : Bool;
   //    res_6335 : Bool;
   //    res_6336 : Bool;
   //    res_6337 : Bool;
   //    mdapdaCoolant : Bool;
   //    mdapdaChipConveyor : Bool;
   //    mdapdaExtraction : Bool;
   //    mdapdaWater : Bool;
   //    mdapdaCompressedAir : Bool;
   //    mdapdaExtinguishingSystem : Bool;
   //    mdaPdaReserve6 : Bool;
   //    mdaPdaReserve7 : Bool;
   //    mdapdaNoPlant1 : Char;
   //    mdapdaNoPlant2 : Char;
   //    mdapdaNoPlant3 : Char;
   //    mdapdaNoPlant4 : Char;
   //    mdapdaNoPlant5 : Char;
   //    mdapdaNoPlant6 : Char;
   //    mdapdaNoPlant7 : Char;
   //    mdapdaNoPlant8 : Char;
   //    mdapdaNoPlant9 : Char;
   //    mdapdaNoPlant10 : Char;
   //    mdapdaNoPlant11 : Char;
   //    mdapdaNoPlant12 : Char;
   //    mdapdaNoPlant13 : Char;
   //    mdapdaNoPlant14 : Char;
   //    mdapdaNoSpindleShaft : Byte;
   //    mdapdaIdentStringWorkpiece : Array[1..36] of Char;
   //    mdapdaIdentStringLoadcarrier : Array[1..36] of Byte;
   //    mdapdaStatus : Byte;
   //    mdapdaCode50FireAlarmSignal : Bool;
   //    mdapdaCode51Extraction : Bool;
   //    mdapdaCode52ChipRemoval : Bool;
   //    mdapdaCode53CompressedAir : Bool;
   //    mdapdaCode54Coolant : Bool;
   //    mdapdaCode55Unloading : Bool;
   //    reserve7236 : Bool;
   //    reserve7237 : Bool;
   //    mdapdaTriggBitOnMPS : Bool;
   //    mdapdaTriggBitOffMPS : Bool;
   //    res7242 : Bool;
   //    res7243 : Bool;
   //    res7244 : Bool;
   //    res7245 : Bool;
   //    res7246 : Bool;
   //    res7247 : Bool;
   //    mdapdaCodeMPS : Byte;
   //    QStop : Bool;
   //    res726p1 : Bool;
   //    res726p2 : Bool;
   //    res726p3 : Bool;
   //    res726p4 : Bool;
   //    res726p5 : Bool;
   //    res726p6 : Bool;
   //    res726p7 : Bool;
   //    mdapdaShiftRegSynchronization : Byte;
   //    mdapdaPartIdSetReport : Array[1..20] of Bool;
   //    res732 : Array[732..737] of Byte;
   //    res738 : Byte;
   //    mdapdaMasterBufferPrealarm : Bool;
   //    mdapdaMasterBufferAlarm : Bool;
   //    mdapdaMasterConnectStatus : Bool;
   //    res7394 : Bool;
   //    res7395 : Bool;
   //    res7396 : Bool;
   //    res7397 : Bool;
   //    res7398 : Bool;
   //    mdapdaStoreWorkpiecetype : Int;
   //    mdapdaStoreResultCode1 : Byte;
   //    mdapdaStoreResultCode2 : Byte;
   //    mdapdaStoreStatus : Byte;
   //    mdapdaStoreLocation : Byte;
   //    mdapdaStoreIdentString : Array[1..36] of Char;
   //    res782 : Array[782..789] of Byte;
   //    mdapdaWithdrawalWorkpiece : Int;
   //    mdapdaWithdrawalResultCode1 : Byte;
   //    mdapdaWithdrawalResultCode2 : Byte;
   //    mdapdaWithdrawalStatus : Byte;
   //    mdapdaWithdrawalLocation : Byte;
   //    mdapdaWithdrawalidentString : Array[1..36] of Char;
   //    res832 : Array[832..839] of Byte;
   //    mdapdaTriggBytePartIdReport : Byte;
   //    mdapdaTriggByteClocking : Byte;
   //    mdapdaTriggBytePartStorage : Byte;
   //    mdapdaTriggBytePartWithdrawal : Byte;
   //    mdapdaTriggByteAssemblyReport : Byte;
   //    mdapdaTriggBytePartIdSetReport : Byte;
   //    mdapdaTriggByteDataCont1 : Byte;
   //    mdapdaTriggByteDataCont2 : Byte;
   //    mdapdaTriggByteDataCont3 : Byte;
   //    mdapdaTriggByteDataCont4 : Byte;
   //    res850 : Array[850..859] of Byte;
   //    mdapdaJobStsBitPartIdReport : Bool;
   //    mdapdaJobStsBitClocking : Bool;
   //    mdapdaJobStsBitPartStorage : Bool;
   //    mdapdaJobStsBitPartWithdrawal : Bool;
   //    mdapdaJobStsBitAssemblyReport : Bool;
   //    mdapdaJobStsBitiPartIdSetReport : Bool;
   //    mdapdaJobStsBitDataCont1 : Bool;
   //    mdapdaJobStsBitDataCont2 : Bool;
   //    mdapdaJobStsBitDataCont3 : Bool;
   //    mdapdaJobStsBitDataCont4 : Bool;
   //    res8612 : Bool;
   //    res8613 : Bool;
   //    res8614 : Bool;
   //    res8615 : Bool;
   //    res8616 : Bool;
   //    res8617 : Bool;
   //    res862 : Array[862..977] of Byte;
   //    res798 : Byte;
   //    mdapdaTriggBitMachineOff : Bool;
   //    mdapdaTriggBitMachineOn : Bool;
   //    res9792 : Bool;
   //    res9793 : Bool;
   //    res9794 : Bool;
   //    res9795 : Bool;
   //    res9796 : Bool;
   //    res9797 : Bool;
   //    mdapdaTriggBitPartStorage : Bool;
   //    mdapdaTriggBitPartWithdrawal : Bool;
   //    mdapdaTriggBitAssemblyReport : Bool;
   //    mdapdaTriggBitiPartIdSetReport : Bool;
   //    mdapdaTriggBitDataCont1 : Bool;
   //    mdapdaTriggBitDataCont2 : Bool;
   //    mdapdaTriggBitDataCont3 : Bool;
   //    mdapdaTriggBitDataCont4 : Bool;
   //    mdapdaStatusInfeedPart1 : Bool;
   //    mdapdaStatusInfeedPart2 : Bool;
   //    mdapdaStatusInfeedPart3 : Bool;
   //    mdapdaStatusInfeedPart4 : Bool;
   //    mdapdaStatusInfeedPart5 : Bool;
   //    mdapdaStatusInfeedPart6 : Bool;
   //    mdapdaStatusInfeedPart7 : Bool;
   //    mdapdaStatusInfeedPart8 : Bool;
   //    mdapdaStatusInfeedPart9 : Bool;
   //    mdapdaStatusInfeedPart10 : Bool;
   //    mdapdaStatusInfeedPart11 : Bool;
   //    mdapdaStatusInfeedPart12 : Bool;
   //    mdapdaStatusInfeedPart13 : Bool;
   //    mdapdaStatusInfeedPart14 : Bool;
   //    mdapdaStatusInfeedPart15 : Bool;
   //    mdapdaStatusInfeedPart16 : Bool;
   //    mdapdaStatusInfeedPart17 : Bool;
   //    mdapdaStatusInfeedPart18 : Bool;
   //    mdapdaStatusInfeedPart19 : Bool;
   //    mdapdaStatusInfeedPart20 : Bool;
   //    mdapdaStatusInfeedPart21 : Bool;
   //    mdapdaStatusInfeedPart22 : Bool;
   //    mdapdaStatusInfeedPart23 : Bool;
   //    mdapdaStatusInfeedPart24 : Bool;
   //    mdapdaStatusInfeedPart25 : Bool;
   //    mdapdaStatusInfeedPart26 : Bool;
   //    mdapdaStatusInfeedPart27 : Bool;
   //    mdapdaStatusInfeedPart28 : Bool;
   //    mdapdaStatusInfeedPart29 : Bool;
   //    mdapdaStatusInfeedPart30 : Bool;
   //    mdapdaStatusInfeedPart31 : Bool;
   //    mdapdaStatusInfeedPart32 : Bool;
   //    mdapdaOverride0 : Bool;
   //    mdapdaManualEndOfToolLife : Bool;
   //    mdapdaManualToolBreakage : Bool;
   //    mdapdaManualWorkpieceQuality : Bool;
   //    mdapdaManualCondMonitoring : Bool;
   //    mdapdaInventoryNoFilter : Bool;
   //    mdapdaLifeHistoryQuery : Bool;
   //    mdapdaManualAcknoledge : Bool;
   //    res_724 : Array[987..1001] of Byte;
   //    workpiecetypeLoadingBelt : Word;
   //    workpiecetypeExitBelt : Word;
   //    cntTotalWorkpieces : DWord;
   //    cntTotalWorkpiecesNotOk : Word;
   //    cntDailyWorkpieces : Word;
   //    cntDailyWorkpiecesNotOk : Word;
   //    cntShiftWorkpieces : Word;
   //    cntShiftWorkpiecesNotOk : Word;
   //    cntWorkpiecetype { S7_SetPoint := 'True'} : Array[1..32] of "LTLP_typeWorkpieceCount";
   //    cycleTimeCompleteMachine : Word;
   //    cycleTime : Array[1..40] of Word;
   //    displayedMachinigUnit : Array[1..42] of Bool;
   //    workpieceTypeStation : Array[1..40] of Struct
   //       workpieceType : Word;
   //       typeAPresent : Bool;
   //       typeAOk : Bool;
   //       typeBPresent : Bool;
   //       typeBOk : Bool;
   //       typeCPresent : Bool;
   //       typeCOk : Bool;
   //       typeDPresent : Bool;
   //       typeDOk : Bool;
   //       typeEPresent : Bool;
   //       typeEOk : Bool;
   //       typeFPresent : Bool;
   //       typeFOk : Bool;
   //       typeGPresent : Bool;
   //       typeGOk : Bool;
   //       typeHPresent : Bool;
   //       typeHOk : Bool;
   //    END_STRUCT;
   //    completionReportUnit1 : Bool;
   //    transportPositionUnit1 : Bool;
   //    faultUnit1 : Bool;
   //    automaticModeUnit1 : Bool;
   //    protectiveDoorsUnit1 : Bool;
   //    unitInOperationUnit1 : Bool;
   //    toolNoReachedUnit1 : Bool;
   //    emergencyStopActUnit1 : Bool;
   //    completionReportUnit2 : Bool;
   //    transportPositionUnit2 : Bool;
   //    faultUnit2 : Bool;
   //    automaticModeUnit2 : Bool;
   //    protectiveDoorsUnit2 : Bool;
   //    unitInOperationUnit2 : Bool;
   //    toolNoReachedUnit2 : Bool;
   //    emergencyStopActUnit2 : Bool;
   //    completionReportUnit3 : Bool;
   //    transportUnitell_Unit3 : Bool;
   //    Unitoerung_Unit3 : Bool;
   //    automaticModeUnit3 : Bool;
   //    protectiveDoorsUnit3 : Bool;
   //    unitInOperationUnit3 : Bool;
   //    toolNoReachedUnit3 : Bool;
   //    emergencyStopActUnit3 : Bool;
   //    completionReportUnit4 : Bool;
   //    transportUnitell_Unit4 : Bool;
   //    Unitoerung_Unit4 : Bool;
   //    automaticModeUnit4 : Bool;
   //    protectiveDoorsUnit4 : Bool;
   //    unitInOperationUnit4 : Bool;
   //    toolNoReachedUnit4 : Bool;
   //    emergencyStopActUnit4 : Bool;
   //    completionReportUnit5 : Bool;
   //    transportUnitell_Unit5 : Bool;
   //    Unitoerung_Unit5 : Bool;
   //    automaticModeUnit5 : Bool;
   //    protectiveDoorsUnit5 : Bool;
   //    unitInOperationUnit5 : Bool;
   //    toolNoReachedUnit5 : Bool;
   //    emergencyStopActUnit5 : Bool;
   //    completionReportUnit6 : Bool;
   //    transportUnitell_Unit6 : Bool;
   //    Unitoerung_Unit6 : Bool;
   //    automaticModeUnit6 : Bool;
   //    protectiveDoorsUnit6 : Bool;
   //    unitInOperationUnit6 : Bool;
   //    toolNoReachedUnit6 : Bool;
   //    emergencyStopActUnit6 : Bool;
   //    completionReportUnit7 : Bool;
   //    transportUnitell_Unit7 : Bool;
   //    Unitoerung_Unit7 : Bool;
   //    automaticModeUnit7 : Bool;
   //    protectiveDoorsUnit7 : Bool;
   //    unitInOperationUnit7 : Bool;
   //    toolNoReachedUnit7 : Bool;
   //    emergencyStopActUnit7 : Bool;
   //    completionReportUnit8 : Bool;
   //    transportUnitell_Unit8 : Bool;
   //    Unitoerung_Unit8 : Bool;
   //    automaticModeUnit8 : Bool;
   //    protectiveDoorsUnit8 : Bool;
   //    unitInOperationUnit8 : Bool;
   //    toolNoReachedUnit8 : Bool;
   //    emergencyStopActUnit8 : Bool;
   //    completionReportUnit9 : Bool;
   //    transportUnitell_Unit9 : Bool;
   //    Unitoerung_Unit9 : Bool;
   //    automaticModeUnit9 : Bool;
   //    protectiveDoorsUnit9 : Bool;
   //    unitInOperationUnit9 : Bool;
   //    toolNoReachedUnit9 : Bool;
   //    emergencyStopActUnit9 : Bool;
   //    completionReportUnit10 : Bool;
   //    transportUnitell_Unit10 : Bool;
   //    Unitoerung_Unit10 : Bool;
   //    automaticModeUnit10 : Bool;
   //    protectiveDoorsUnit10 : Bool;
   //    unitInOperationUnit10 : Bool;
   //    toolNoReachedUnit10 : Bool;
   //    emergencyStopActUnit10 : Bool;
   //    completionReportUnit11 : Bool;
   //    transportUnitell_Unit11 : Bool;
   //    Unitoerung_Unit11 : Bool;
   //    automaticModeUnit11 : Bool;
   //    protectiveDoorsUnit11 : Bool;
   //    unitInOperationUnit11 : Bool;
   //    toolNoReachedUnit11 : Bool;
   //    emergencyStopActUnit11 : Bool;
   //    completionReportUnit12 : Bool;
   //    transportUnitell_Unit12 : Bool;
   //    Unitoerung_Unit12 : Bool;
   //    automaticModeUnit12 : Bool;
   //    protectiveDoorsUnit12 : Bool;
   //    unitInOperationUnit12 : Bool;
   //    toolNoReachedUnit12 : Bool;
   //    emergencyStopActUnit12 : Bool;
   //    completionReportUnit13 : Bool;
   //    transportUnitell_Unit13 : Bool;
   //    Unitoerung_Unit13 : Bool;
   //    automaticModeUnit13 : Bool;
   //    protectiveDoorsUnit13 : Bool;
   //    unitInOperationUnit13 : Bool;
   //    toolNoReachedUnit13 : Bool;
   //    emergencyStopActUnit13 : Bool;
   //    completionReportUnit14 : Bool;
   //    transportUnitell_Unit14 : Bool;
   //    Unitoerung_Unit14 : Bool;
   //    automaticModeUnit14 : Bool;
   //    protectiveDoorsUnit14 : Bool;
   //    unitInOperationUnit14 : Bool;
   //    toolNoReachedUnit14 : Bool;
   //    emergencyStopActUnit14 : Bool;
   //    completionReportUnit15 : Bool;
   //    transportUnitell_Unit15 : Bool;
   //    Unitoerung_Unit15 : Bool;
   //    automaticModeUnit15 : Bool;
   //    protectiveDoorsUnit15 : Bool;
   //    unitInOperationUnit15 : Bool;
   //    toolNoReachedUnit15 : Bool;
   //    emergencyStopActUnit15 : Bool;
   //    completionReportUnit16 : Bool;
   //    transportUnitell_Unit16 : Bool;
   //    Unitoerung_Unit16 : Bool;
   //    automaticModeUnit16 : Bool;
   //    protectiveDoorsUnit16 : Bool;
   //    unitInOperationUnit16 : Bool;
   //    toolNoReachedUnit16 : Bool;
   //    emergencyStopActUnit16 : Bool;
   //    completionReportUnit17 : Bool;
   //    transportUnitell_Unit17 : Bool;
   //    Unitoerung_Unit17 : Bool;
   //    automaticModeUnit17 : Bool;
   //    protectiveDoorsUnit17 : Bool;
   //    unitInOperationUnit17 : Bool;
   //    toolNoReachedUnit17 : Bool;
   //    emergencyStopActUnit17 : Bool;
   //    completionReportUnit18 : Bool;
   //    transportUnitell_Unit18 : Bool;
   //    Unitoerung_Unit18 : Bool;
   //    automaticModeUnit18 : Bool;
   //    protectiveDoorsUnit18 : Bool;
   //    unitInOperationUnit18 : Bool;
   //    toolNoReachedUnit18 : Bool;
   //    emergencyStopActUnit18 : Bool;
   //    completionReportUnit19 : Bool;
   //    transportUnitell_Unit19 : Bool;
   //    Unitoerung_Unit19 : Bool;
   //    automaticModeUnit19 : Bool;
   //    protectiveDoorsUnit19 : Bool;
   //    unitInOperationUnit19 : Bool;
   //    toolNoReachedUnit19 : Bool;
   //    emergencyStopActUnit19 : Bool;
   //    completionReportUnit20 : Bool;
   //    transportUnitell_Unit20 : Bool;
   //    Unitoerung_Unit20 : Bool;
   //    automaticModeUnit20 : Bool;
   //    protectiveDoorsUnit20 : Bool;
   //    unitInOperationUnit20 : Bool;
   //    toolNoReachedUnit20 : Bool;
   //    emergencyStopActUnit20 : Bool;
   //    completionReportUnit21 : Bool;
   //    transportUnitell_Unit21 : Bool;
   //    Unitoerung_Unit21 : Bool;
   //    automaticModeUnit21 : Bool;
   //    protectiveDoorsUnit21 : Bool;
   //    unitInOperationUnit21 : Bool;
   //    toolNoReachedUnit21 : Bool;
   //    emergencyStopActUnit21 : Bool;
   //    completionReportUnit22 : Bool;
   //    transportUnitell_Unit22 : Bool;
   //    Unitoerung_Unit22 : Bool;
   //    automaticModeUnit22 : Bool;
   //    protectiveDoorsUnit22 : Bool;
   //    unitInOperationUnit22 : Bool;
   //    toolNoReachedUnit22 : Bool;
   //    emergencyStopActUnit22 : Bool;
   //    completionReportUnit23 : Bool;
   //    transportUnitell_Unit23 : Bool;
   //    Unitoerung_Unit23 : Bool;
   //    automaticModeUnit23 : Bool;
   //    protectiveDoorsUnit23 : Bool;
   //    unitInOperationUnit23 : Bool;
   //    toolNoReachedUnit23 : Bool;
   //    emergencyStopActUnit23 : Bool;
   //    completionReportUnit24 : Bool;
   //    transportUnitell_Unit24 : Bool;
   //    Unitoerung_Unit24 : Bool;
   //    automaticModeUnit24 : Bool;
   //    protectiveDoorsUnit24 : Bool;
   //    unitInOperationUnit24 : Bool;
   //    toolNoReachedUnit24 : Bool;
   //    emergencyStopActUnit24 : Bool;
   //    completionReportUnit25 : Bool;
   //    transportUnitell_Unit25 : Bool;
   //    Unitoerung_Unit25 : Bool;
   //    automaticModeUnit25 : Bool;
   //    protectiveDoorsUnit25 : Bool;
   //    unitInOperationUnit25 : Bool;
   //    toolNoReachedUnit25 : Bool;
   //    emergencyStopActUnit25 : Bool;
   //    completionReportUnit26 : Bool;
   //    transportUnitell_Unit26 : Bool;
   //    Unitoerung_Unit26 : Bool;
   //    automaticModeUnit26 : Bool;
   //    protectiveDoorsUnit26 : Bool;
   //    unitInOperationUnit26 : Bool;
   //    toolNoReachedUnit26 : Bool;
   //    emergencyStopActUnit26 : Bool;
   //    completionReportUnit27 : Bool;
   //    transportUnitell_Unit27 : Bool;
   //    Unitoerung_Unit27 : Bool;
   //    automaticModeUnit27 : Bool;
   //    protectiveDoorsUnit27 : Bool;
   //    unitInOperationUnit27 : Bool;
   //    toolNoReachedUnit27 : Bool;
   //    emergencyStopActUnit27 : Bool;
   //    completionReportUnit28 : Bool;
   //    transportUnitell_Unit28 : Bool;
   //    Unitoerung_Unit28 : Bool;
   //    automaticModeUnit28 : Bool;
   //    protectiveDoorsUnit28 : Bool;
   //    unitInOperationUnit28 : Bool;
   //    toolNoReachedUnit28 : Bool;
   //    emergencyStopActUnit28 : Bool;
   //    completionReportUnit29 : Bool;
   //    transportUnitell_Unit29 : Bool;
   //    Unitoerung_Unit29 : Bool;
   //    automaticModeUnit29 : Bool;
   //    protectiveDoorsUnit29 : Bool;
   //    unitInOperationUnit29 : Bool;
   //    toolNoReachedUnit29 : Bool;
   //    emergencyStopActUnit29 : Bool;
   //    completionReportUnit30 : Bool;
   //    transportUnitell_Unit30 : Bool;
   //    Unitoerung_Unit30 : Bool;
   //    automaticModeUnit30 : Bool;
   //    protectiveDoorsUnit30 : Bool;
   //    unitInOperationUnit30 : Bool;
   //    toolNoReachedUnit30 : Bool;
   //    emergencyStopActUnit30 : Bool;
   //    completionReportUnit31 : Bool;
   //    transportUnitell_Unit31 : Bool;
   //    Unitoerung_Unit31 : Bool;
   //    automaticModeUnit31 : Bool;
   //    protectiveDoorsUnit31 : Bool;
   //    unitInOperationUnit31 : Bool;
   //    toolNoReachedUnit31 : Bool;
   //    emergencyStopActUnit31 : Bool;
   //    completionReportUnit32 : Bool;
   //    transportUnitell_Unit32 : Bool;
   //    Unitoerung_Unit32 : Bool;
   //    automaticModeUnit32 : Bool;
   //    protectiveDoorsUnit32 : Bool;
   //    unitInOperationUnit32 : Bool;
   //    toolNoReachedUnit32 : Bool;
   //    emergencyStopActUnit32 : Bool;
   //    completionReportUnit33 : Bool;
   //    transportUnitell_Unit33 : Bool;
   //    Unitoerung_Unit33 : Bool;
   //    automaticModeUnit33 : Bool;
   //    protectiveDoorsUnit33 : Bool;
   //    unitInOperationUnit33 : Bool;
   //    toolNoReachedUnit33 : Bool;
   //    emergencyStopActUnit33 : Bool;
   //    completionReportUnit34 : Bool;
   //    transportUnitell_Unit34 : Bool;
   //    Unitoerung_Unit34 : Bool;
   //    automaticModeUnit34 : Bool;
   //    protectiveDoorsUnit34 : Bool;
   //    unitInOperationUnit34 : Bool;
   //    toolNoReachedUnit34 : Bool;
   //    emergencyStopActUnit34 : Bool;
   //    completionReportUnit35 : Bool;
   //    transportUnitell_Unit35 : Bool;
   //    Unitoerung_Unit35 : Bool;
   //    automaticModeUnit35 : Bool;
   //    protectiveDoorsUnit35 : Bool;
   //    unitInOperationUnit35 : Bool;
   //    toolNoReachedUnit35 : Bool;
   //    emergencyStopActUnit35 : Bool;
   //    completionReportUnit36 : Bool;
   //    transportUnitell_Unit36 : Bool;
   //    Unitoerung_Unit36 : Bool;
   //    automaticModeUnit36 : Bool;
   //    protectiveDoorsUnit36 : Bool;
   //    unitInOperationUnit36 : Bool;
   //    toolNoReachedUnit36 : Bool;
   //    emergencyStopActUnit36 : Bool;
   //    completionReportUnit37 : Bool;
   //    transportUnitell_Unit37 : Bool;
   //    Unitoerung_Unit37 : Bool;
   //    automaticModeUnit37 : Bool;
   //    protectiveDoors : Bool;
   //    unitInOperationUnit37 : Bool;
   //    toolNoReachedUnit37 : Bool;
   //    emergencyStopActUnit37 : Bool;
   //    completionReportUnit38 : Bool;
   //    transportUnitell_Unit38 : Bool;
   //    Unitoerung_Unit38 : Bool;
   //    automaticModeUnit38 : Bool;
   //    protectiveDoorsUnit38 : Bool;
   //    unitInOperationUnit38 : Bool;
   //    toolNoReachedUnit38 : Bool;
   //    emergencyStopActUnit38 : Bool;
   //    completionReportUnit39 : Bool;
   //    transportUnitell_Unit39 : Bool;
   //    Unitoerung_Unit39 : Bool;
   //    automaticModeUnit39 : Bool;
   //    protectiveDoorsUnit39 : Bool;
   //    unitInOperationUnit39 : Bool;
   //    toolNoReachedUnit39 : Bool;
   //    emergencyStopActUnit39 : Bool;
   //    completionReportUnit40 : Bool;
   //    transportUnitell_Unit40 : Bool;
   //    Unitoerung_Unit40 : Bool;
   //    automaticModeUnit40 : Bool;
   //    protectiveDoorsUnit40 : Bool;
   //    unitInOperationUnit40 : Bool;
   //    toolNoReachedUnit40 : Bool;
   //    emergencyStopActUnit40 : Bool;
   //    clampedUnit1 : Bool;
   //    releasedUnit1 : Bool;
   //    partClampedUnit1 : Bool;
   //    partReleasedUnit1 : Bool;
   //    clampedUnit2 : Bool;
   //    releasedUnit2 : Bool;
   //    partClampedUnit2 : Bool;
   //    partReleasedUnit2 : Bool;
   //    clampedUnit3 : Bool;
   //    releasedUnit3 : Bool;
   //    partClampedUnit3 : Bool;
   //    partReleasedUnit3 : Bool;
   //    clampedUnit4 : Bool;
   //    releasedUnit4 : Bool;
   //    partClampedUnit4 : Bool;
   //    partReleasedUnit4 : Bool;
   //    clampedUnit5 : Bool;
   //    releasedUnit5 : Bool;
   //    partClampedUnit5 : Bool;
   //    partReleasedUnit5 : Bool;
   //    clampedUnit6 : Bool;
   //    releasedUnit6 : Bool;
   //    partClampedUnit6 : Bool;
   //    partReleasedUnit6 : Bool;
   //    clampedUnit7 : Bool;
   //    releasedUnit7 : Bool;
   //    partClampedUnit7 : Bool;
   //    partReleasedUnit7 : Bool;
   //    clampedUnit8 : Bool;
   //    releasedUnit8 : Bool;
   //    partClampedUnit8 : Bool;
   //    partReleasedUnit8 : Bool;
   //    clampedUnit9 : Bool;
   //    releasedUnit9 : Bool;
   //    partClampedUnit9 : Bool;
   //    partReleasedUnit9 : Bool;
   //    clampedUnit10 : Bool;
   //    releasedUnit10 : Bool;
   //    partClampedUnit10 : Bool;
   //    partReleasedUnit10 : Bool;
   //    clampedUnit11 : Bool;
   //    releasedUnit11 : Bool;
   //    partClampedUnit11 : Bool;
   //    partReleasedUnit11 : Bool;
   //    clampedUnit12 : Bool;
   //    releasedUnit12 : Bool;
   //    partClampedUnit12 : Bool;
   //    partReleasedUnit12 : Bool;
   //    clampedUnit13 : Bool;
   //    releasedUnit13 : Bool;
   //    partClampedUnit13 : Bool;
   //    partReleasedUnit13 : Bool;
   //    clampedUnit14 : Bool;
   //    releasedUnit14 : Bool;
   //    partClampedUnit14 : Bool;
   //    partReleasedUnit14 : Bool;
   //    clampedUnit15 : Bool;
   //    releasedUnit15 : Bool;
   //    partClampedUnit15 : Bool;
   //    partReleasedUnit15 : Bool;
   //    clampedUnit16 : Bool;
   //    releasedUnit16 : Bool;
   //    partClampedUnit16 : Bool;
   //    partReleasedUnit16 : Bool;
   //    clampedUnit17 : Bool;
   //    releasedUnit17 : Bool;
   //    partClampedUnit17 : Bool;
   //    partReleasedUnit17 : Bool;
   //    clampedUnit18 : Bool;
   //    releasedUnit18 : Bool;
   //    partClampedUnit18 : Bool;
   //    partReleasedUnit18 : Bool;
   //    clampedUnit19 : Bool;
   //    releasedUnit19 : Bool;
   //    partClampedUnit19 : Bool;
   //    partReleasedUnit19 : Bool;
   //    clampedUnit20 : Bool;
   //    releasedUnit20 : Bool;
   //    partClampedUnit20 : Bool;
   //    partReleasedUnit20 : Bool;
   //    clampedUnit21 : Bool;
   //    releasedUnit21 : Bool;
   //    partClampedUnit21 : Bool;
   //    partReleasedUnit21 : Bool;
   //    clampedUnit22 : Bool;
   //    releasedUnit22 : Bool;
   //    partClampedUnit22 : Bool;
   //    partReleasedUnit22 : Bool;
   //    clampedUnit23 : Bool;
   //    releasedUnit23 : Bool;
   //    partClampedUnit23 : Bool;
   //    partReleasedUnit23 : Bool;
   //    clampedUnit24 : Bool;
   //    releasedUnit24 : Bool;
   //    partClampedUnit24 : Bool;
   //    partReleasedUnit24 : Bool;
   //    clampedUnit25 : Bool;
   //    releasedUnit25 : Bool;
   //    partClampedUnit25 : Bool;
   //    partReleasedUnit25 : Bool;
   //    clampedUnit26 : Bool;
   //    releasedUnit26 : Bool;
   //    partClampedUnit26 : Bool;
   //    partReleasedUnit26 : Bool;
   //    clampedUnit27 : Bool;
   //    releasedUnit27 : Bool;
   //    partClampedUnit27 : Bool;
   //    partReleasedUnit27 : Bool;
   //    clampedUnit28 : Bool;
   //    releasedUnit28 : Bool;
   //    partClampedUnit28 : Bool;
   //    partReleasedUnit28 : Bool;
   //    clampedUnit29 : Bool;
   //    releasedUnit29 : Bool;
   //    partClampedUnit29 : Bool;
   //    partReleasedUnit29 : Bool;
   //    clampedUnit30 : Bool;
   //    releasedUnit30 : Bool;
   //    partClampedUnit30 : Bool;
   //    partReleasedUnit30 : Bool;
   //    clampedUnit31 : Bool;
   //    releasedUnit31 : Bool;
   //    partClampedUnit31 : Bool;
   //    partReleasedUnit31 : Bool;
   //    clampedUnit32 : Bool;
   //    releasedUnit32 : Bool;
   //    partClampedUnit32 : Bool;
   //    partReleasedUnit32 : Bool;
   //    clampedUnit33 : Bool;
   //    releasedUnit33 : Bool;
   //    partClampedUnit33 : Bool;
   //    partReleasedUnit33 : Bool;
   //    clampedUnit34 : Bool;
   //    releasedUnit34 : Bool;
   //    partClampedUnit34 : Bool;
   //    partReleasedUnit34 : Bool;
   //    clampedUnit35 : Bool;
   //    releasedUnit35 : Bool;
   //    partClampedUnit35 : Bool;
   //    partReleasedUnit35 : Bool;
   //    clampedUnit36 : Bool;
   //    releasedUnit36 : Bool;
   //    partClampedUnit36 : Bool;
   //    partReleasedUnit36 : Bool;
   //    clampedUnit37 : Bool;
   //    releasedUnit37 : Bool;
   //    partClampedUnit37 : Bool;
   //    partReleasedUnit37 : Bool;
   //    clampedUnit38 : Bool;
   //    releasedUnit38 : Bool;
   //    partClampedUnit38 : Bool;
   //    partReleasedUnit38 : Bool;
   //    clampedUnit39 : Bool;
   //    releasedUnit39 : Bool;
   //    partClampedUnit39 : Bool;
   //    partReleasedUnit39 : Bool;
   //    clampedUnit40 : Bool;
   //    releasedUnit40 : Bool;
   //    partClampedUnit40 : Bool;
   //    partReleasedUnit40 : Bool;
   //    infeedOccupied : Bool;
   //    infeedEmpty : Bool;
   //    exitFree : Bool;
   //    exitOccupied : Bool;
   //    limitedFeed1Open : Bool;
   //    limitedFeed1Closed : Bool;
   //    limitedFeed2Open : Bool;
   //    limitedFeed2Closed : Bool;
   //    limitedFeed3Open : Bool;
   //    limitedFeed3Closed : Bool;
   //    limitedFeed4Open : Bool;
   //    limitedFeed4Closed : Bool;
   //    limitedFeed5Open : Bool;
   //    limitedFeed5Closed : Bool;
   //    limitedFeed6Open : Bool;
   //    limitedFeed6Closed : Bool;
   //    transferBarIntermedPosition : Bool;
   //    res_111 : Bool;
   //    res_12 : Bool;
   //    res_13 : Bool;
   //    transferBar1Front : Bool;
   //    transferBar1Rear : Bool;
   //    transferBar1Bottom : Bool;
   //    transferBar1Top : Bool;
   //    transferBar2IntermedPosition : Bool;
   //    res_14 : Bool;
   //    res_15 : Bool;
   //    res_16 : Bool;
   //    transferBar2Front : Bool;
   //    transferBar2Rear : Bool;
   //    transferBar2Bottom : Bool;
   //    transferBar2Top : Bool;
   //    powerupCondOn1 : Bool;
   //    powerupCondOff1 : Bool;
   //    powerupCondOn2 : Bool;
   //    powerupCondOff2 : Bool;
   //    powerupCondOn3 : Bool;
   //    powerupCondOff3 : Bool;
   //    powerupCondOn4 : Bool;
   //    powerupCondOff4 : Bool;
   //    powerupCondOn5 : Bool;
   //    powerupCondOff5 : Bool;
   //    powerupCondOn6 : Bool;
   //    powerupCondOff6 : Bool;
   //    powerupCondOn7 : Bool;
   //    powerupCondOff7 : Bool;
   //    powerupCondOn8 : Bool;
   //    powerupCondOff8 : Bool;
   //    powerupCondOn9 : Bool;
   //    powerupCondOff9 : Bool;
   //    powerupCondOn10 : Bool;
   //    powerupCondOff10 : Bool;
   //    powerupCondOn11 : Bool;
   //    powerupCondOff11 : Bool;
   //    powerupCondOn12 : Bool;
   //    powerupCondOff12 : Bool;
   //    powerupCondOn13 : Bool;
   //    powerupCondOff13 : Bool;
   //    powerupCondOn14 : Bool;
   //    powerupCondOff14 : Bool;
   //    powerupCondOn15 : Bool;
   //    powerupCondOff15 : Bool;
   //    powerupCondOn16 : Bool;
   //    powerupCondOff16 : Bool;
   //    powerupCondOn17 : Bool;
   //    powerupCondOff17 : Bool;
   //    powerupCondOn18 : Bool;
   //    powerupCondOff18 : Bool;
   //    powerupCondOn19 : Bool;
   //    powerupCondOff19 : Bool;
   //    powerupCondOn20 : Bool;
   //    powerupCondOff20 : Bool;
   //    powerupCondOn21 : Bool;
   //    powerupCondOff21 : Bool;
   //    powerupCondOn22 : Bool;
   //    powerupCondOff22 : Bool;
   //    powerupCondOn23 : Bool;
   //    powerupCondOff23 : Bool;
   //    powerupCondOn24 : Bool;
   //    powerupCondOff24 : Bool;
   //    powerupCondOn25 : Bool;
   //    powerupCondOff25 : Bool;
   //    powerupCondOn26 : Bool;
   //    powerupCondOff26 : Bool;
   //    powerupCondOn27 : Bool;
   //    powerupCondOff27 : Bool;
   //    powerupCondOn28 : Bool;
   //    powerupCondOff28 : Bool;
   //    powerupCondOn29 : Bool;
   //    powerupCondOff29 : Bool;
   //    powerupCondOn30 : Bool;
   //    powerupCondOff30 : Bool;
   //    powerupCondOn31 : Bool;
   //    powerupCondOff31 : Bool;
   //    powerupCondOn32 : Bool;
   //    powerupCondOff32 : Bool;
   //    powerupCondOn33 : Bool;
   //    powerupCondOff33 : Bool;
   //    powerupCondOn34 : Bool;
   //    powerupCondOff34 : Bool;
   //    powerupCondOn35 : Bool;
   //    powerupCondOff35 : Bool;
   //    powerupCondOn36 : Bool;
   //    powerupCondOff36 : Bool;
   //    powerupCondOn37 : Bool;
   //    powerupCondOff37 : Bool;
   //    powerupCondOn38 : Bool;
   //    powerupCondOff38 : Bool;
   //    powerupCondOn39 : Bool;
   //    powerupCondOff39 : Bool;
   //    powerupCondOn40 : Bool;
   //    powerupCondOff40 : Bool;
   //    powerupCondOn41 : Bool;
   //    powerupCondOff41 : Bool;
   //    powerupCondOn42 : Bool;
   //    powerupCondOff42 : Bool;
   //    powerupCondOn43 : Bool;
   //    powerupCondOff43 : Bool;
   //    powerupCondOn44 : Bool;
   //    powerupCondOff44 : Bool;
   //    powerupCondOn45 : Bool;
   //    powerupCondOff45 : Bool;
   //    powerupCondOn46 : Bool;
   //    powerupCondOff46 : Bool;
   //    powerupCondOn47 : Bool;
   //    powerupCondOff47 : Bool;
   //    powerupCondOn48 : Bool;
   //    powerupCondOff48 : Bool;
   //    groupDeselection : Array[1..40] of Bool;
   //    res1 : Array[1798..1804] of Byte;
   //    nutRun1NotMachined : Bool;
   //    nutRun1Ok : Bool;
   //    nutRun1NotOk : Bool;
   //    nutRun1Reserve : Bool;
   //    nutRun1TorqueHigh : Bool;
   //    nutRun1TorqueLow : Bool;
   //    nutRun1AngleHigh : Bool;
   //    nutRun1AngleLow : Bool;
   //    nutRun2NotMachined : Bool;
   //    nutRun2Ok : Bool;
   //    nutRun2NotOk : Bool;
   //    nutRun2Reserve : Bool;
   //    nutRun2TorqueHigh : Bool;
   //    nutRun2TorqueLow : Bool;
   //    nutRun2AngleHigh : Bool;
   //    nutRun2AngleLow : Bool;
   //    nutRun3NotMachined : Bool;
   //    nutRun3Ok : Bool;
   //    nutRun3NotOk : Bool;
   //    nutRun3Reserve : Bool;
   //    nutRun3TorqueHigh : Bool;
   //    nutRun3TorqueLow : Bool;
   //    nutRun3AngleHigh : Bool;
   //    nutRun3AngleLow : Bool;
   //    nutRun4NotMachined : Bool;
   //    nutRun4Ok : Bool;
   //    nutRun4NotOk : Bool;
   //    nutRun4Reserve : Bool;
   //    nutRun4TorqueHigh : Bool;
   //    nutRun4TorqueLow : Bool;
   //    nutRun4AngleHigh : Bool;
   //    nutRun4AngleLow : Bool;
   //    nutRun5NotMachined : Bool;
   //    nutRun5Ok : Bool;
   //    nutRun5NotOk : Bool;
   //    nutRun5Reserve : Bool;
   //    nutRun5TorqueHigh : Bool;
   //    nutRun5TorqueLow : Bool;
   //    nutRun5AngleHigh : Bool;
   //    nutRun5AngleLow : Bool;
   //    nutRun6NotMachined : Bool;
   //    nutRun6Ok : Bool;
   //    nutRun6NotOk : Bool;
   //    nutRun6Reserve : Bool;
   //    nutRun6TorqueHigh : Bool;
   //    nutRun6TorqueLow : Bool;
   //    nutRun6AngleHigh : Bool;
   //    nutRun6AngleLow : Bool;
   //    nutRun7NotMachined : Bool;
   //    nutRun7Ok : Bool;
   //    nutRun7NotOk : Bool;
   //    nutRun7Reserve : Bool;
   //    nutRun7TorqueHigh : Bool;
   //    nutRun7TorqueLow : Bool;
   //    nutRun7AngleHigh : Bool;
   //    nutRun7AngleLow : Bool;
   //    nutRun8NotMachined : Bool;
   //    nutRun8Ok : Bool;
   //    nutRun8NotOk : Bool;
   //    nutRun8Reserve : Bool;
   //    nutRun8TorqueHigh : Bool;
   //    nutRun8TorqueLow : Bool;
   //    nutRun8AngleHigh : Bool;
   //    nutRun8AngleLow : Bool;
   //    nutRun9NotMachined : Bool;
   //    nutRun9Ok : Bool;
   //    nutRun9NotOk : Bool;
   //    nutRun9Reserve : Bool;
   //    nutRun9TorqueHigh : Bool;
   //    nutRun9TorqueLow : Bool;
   //    nutRun9AngleHigh : Bool;
   //    nutRun9AngleLow : Bool;
   //    nutRun10NotMachined : Bool;
   //    nutRun10Ok : Bool;
   //    nutRun10NotOk : Bool;
   //    nutRun10Reserve : Bool;
   //    nutRun10TorqueHigh : Bool;
   //    nutRun10TorqueLow : Bool;
   //    nutRun10AngleHigh : Bool;
   //    nutRun10AngleLow : Bool;
   //    nutRun11NotMachined : Bool;
   //    nutRun11Ok : Bool;
   //    nutRun11NotOk : Bool;
   //    nutRun11Reserve : Bool;
   //    nutRun11TorqueHigh : Bool;
   //    nutRun11TorqueLow : Bool;
   //    nutRun11AngleHigh : Bool;
   //    nutRun11AngleLow : Bool;
   //    nutRun12NotMachined : Bool;
   //    nutRun12Ok : Bool;
   //    nutRun12NotOk : Bool;
   //    nutRun12Reserve : Bool;
   //    nutRun12TorqueHigh : Bool;
   //    nutRun12TorqueLow : Bool;
   //    nutRun12AngleHigh : Bool;
   //    nutRun12AngleLow : Bool;
   //    nutRun13NotMachined : Bool;
   //    nutRun13Ok : Bool;
   //    nutRun13NotOk : Bool;
   //    nutRun13Reserve : Bool;
   //    nutRun13TorqueHigh : Bool;
   //    nutRun13TorqueLow : Bool;
   //    nutRun13AngleHigh : Bool;
   //    nutRun13AngleLow : Bool;
   //    nutRun14NotMachined : Bool;
   //    nutRun14Ok : Bool;
   //    nutRun14NotOk : Bool;
   //    nutRun14Reserve : Bool;
   //    nutRun14TorqueHigh : Bool;
   //    nutRun14TorqueLow : Bool;
   //    nutRun14AngleHigh : Bool;
   //    nutRun14AngleLow : Bool;
   //    nutRun15NotMachined : Bool;
   //    nutRun15Ok : Bool;
   //    nutRun15NotOk : Bool;
   //    nutRun15Reserve : Bool;
   //    nutRun15TorqueHigh : Bool;
   //    nutRun15TorqueLow : Bool;
   //    nutRun15AngleHigh : Bool;
   //    nutRun15AngleLow : Bool;
   //    nutRun16NotMachined : Bool;
   //    nutRun16Ok : Bool;
   //    nutRun16NotOk : Bool;
   //    nutRun16Reserve : Bool;
   //    nutRun16TorqueHigh : Bool;
   //    nutRun16TorqueLow : Bool;
   //    nutRun16AngleHigh : Bool;
   //    nutRun16AngleLow : Bool;
   //    nutRun17NotMachined : Bool;
   //    nutRun17Ok : Bool;
   //    nutRun17NotOk : Bool;
   //    nutRun17Reserve : Bool;
   //    nutRun17TorqueHigh : Bool;
   //    nutRun17TorqueLow : Bool;
   //    nutRun17AngleHigh : Bool;
   //    nutRun17AngleLow : Bool;
   //    nutRun18NotMachined : Bool;
   //    nutRun18Ok : Bool;
   //    nutRun18NotOk : Bool;
   //    nutRun18Reserve : Bool;
   //    nutRun18TorqueHigh : Bool;
   //    nutRun18TorqueLow : Bool;
   //    nutRun18AngleHigh : Bool;
   //    nutRun18AngleLow : Bool;
   //    nutRun19NotMachined : Bool;
   //    nutRun19Ok : Bool;
   //    nutRun19NotOk : Bool;
   //    nutRun19Reserve : Bool;
   //    nutRun19TorqueHigh : Bool;
   //    nutRun19TorqueLow : Bool;
   //    nutRun19AngleHigh : Bool;
   //    nutRun19AngleLow : Bool;
   //    nutRun20NotMachined : Bool;
   //    nutRun20Ok : Bool;
   //    nutRun20NotOk : Bool;
   //    nutRun20Reserve : Bool;
   //    nutRun20TorqueHigh : Bool;
   //    nutRun20TorqueLow : Bool;
   //    nutRun20AngleHigh : Bool;
   //    nutRun20AngleLow : Bool;
   //    nutRun21NotMachined : Bool;
   //    nutRun21Ok : Bool;
   //    nutRun21NotOk : Bool;
   //    nutRun21Reserve : Bool;
   //    nutRun21TorqueHigh : Bool;
   //    nutRun21TorqueLow : Bool;
   //    nutRun21AngleHigh : Bool;
   //    nutRun21AngleLow : Bool;
   //    nutRun22NotMachined : Bool;
   //    nutRun22Ok : Bool;
   //    nutRun22NotOk : Bool;
   //    nutRun22Reserve : Bool;
   //    nutRun22TorqueHigh : Bool;
   //    nutRun22TorqueLow : Bool;
   //    nutRun22AngleHigh : Bool;
   //    nutRun22AngleLow : Bool;
   //    nutRun23NotMachined : Bool;
   //    nutRun23Ok : Bool;
   //    nutRun23NotOk : Bool;
   //    nutRun23Reserve : Bool;
   //    nutRun23TorqueHigh : Bool;
   //    nutRun23TorqueLow : Bool;
   //    nutRun23AngleHigh : Bool;
   //    nutRun23AngleLow : Bool;
   //    nutRun24NotMachined : Bool;
   //    nutRun24Ok : Bool;
   //    nutRun24NotOk : Bool;
   //    nutRun24Reserve : Bool;
   //    nutRun24TorqueHigh : Bool;
   //    nutRun24TorqueLow : Bool;
   //    nutRun24AngleHigh : Bool;
   //    nutRun24AngleLow : Bool;
   //    nutRun25NotMachined : Bool;
   //    nutRun25Ok : Bool;
   //    nutRun25NotOk : Bool;
   //    nutRun25Reserve : Bool;
   //    nutRun25TorqueHigh : Bool;
   //    nutRun25TorqueLow : Bool;
   //    nutRun25AngleHigh : Bool;
   //    nutRun25AngleLow : Bool;
   //    nutRun26NotMachined : Bool;
   //    nutRun26Ok : Bool;
   //    nutRun26NotOk : Bool;
   //    nutRun26Reserve : Bool;
   //    nutRun26TorqueHigh : Bool;
   //    nutRun26TorqueLow : Bool;
   //    nutRun26AngleHigh : Bool;
   //    nutRun26AngleLow : Bool;
   //    nutRun27NotMachined : Bool;
   //    nutRun27Ok : Bool;
   //    nutRun27NotOk : Bool;
   //    nutRun27Reserve : Bool;
   //    nutRun27TorqueHigh : Bool;
   //    nutRun27TorqueLow : Bool;
   //    nutRun27AngleHigh : Bool;
   //    nutRun27AngleLow : Bool;
   //    nutRun28NotMachined : Bool;
   //    nutRun28Ok : Bool;
   //    nutRun28NotOk : Bool;
   //    nutRun28Reserve : Bool;
   //    nutRun28TorqueHigh : Bool;
   //    nutRun28TorqueLow : Bool;
   //    nutRun28AngleHigh : Bool;
   //    nutRun28AngleLow : Bool;
   //    nutRun29NotMachined : Bool;
   //    nutRun29Ok : Bool;
   //    nutRun29NotOk : Bool;
   //    nutRun29Reserve : Bool;
   //    nutRun29TorqueHigh : Bool;
   //    nutRun29TorqueLow : Bool;
   //    nutRun29AngleHigh : Bool;
   //    nutRun29AngleLow : Bool;
   //    nutRun30NotMachined : Bool;
   //    nutRun30Ok : Bool;
   //    nutRun30NotOk : Bool;
   //    nutRun30Reserve : Bool;
   //    nutRun30TorqueHigh : Bool;
   //    nutRun30TorqueLow : Bool;
   //    nutRun30AngleHigh : Bool;
   //    nutRun30AngleLow : Bool;
   //    nutRun31NotMachined : Bool;
   //    nutRun31Ok : Bool;
   //    nutRun31NotOk : Bool;
   //    nutRun31Reserve : Bool;
   //    nutRun31TorqueHigh : Bool;
   //    nutRun31TorqueLow : Bool;
   //    nutRun31AngleHigh : Bool;
   //    nutRun31AngleLow : Bool;
   //    nutRun32NotMachined : Bool;
   //    nutRun32Ok : Bool;
   //    nutRun32NotOk : Bool;
   //    nutRun32Reserve : Bool;
   //    nutRun32TorqueHigh : Bool;
   //    nutRun32TorqueLow : Bool;
   //    nutRun32AngleHigh : Bool;
   //    nutRun32AngleLow : Bool;
   //    nutRun33NotMachined : Bool;
   //    nutRun33Ok : Bool;
   //    nutRun33NotOk : Bool;
   //    nutRun33Reserve : Bool;
   //    nutRun33TorqueHigh : Bool;
   //    nutRun33TorqueLow : Bool;
   //    nutRun33AngleHigh : Bool;
   //    nutRun33AngleLow : Bool;
   //    nutRun34NotMachined : Bool;
   //    nutRun34Ok : Bool;
   //    nutRun34NotOk : Bool;
   //    nutRun34Reserve : Bool;
   //    nutRun34TorqueHigh : Bool;
   //    nutRun34TorqueLow : Bool;
   //    nutRun34AngleHigh : Bool;
   //    nutRun34AngleLow : Bool;
   //    nutRun35NotMachined : Bool;
   //    nutRun35Ok : Bool;
   //    nutRun35NotOk : Bool;
   //    nutRun35Reserve : Bool;
   //    nutRun35TorqueHigh : Bool;
   //    nutRun35TorqueLow : Bool;
   //    nutRun35AngleHigh : Bool;
   //    nutRun35AngleLow : Bool;
   //    nutRun36NotMachined : Bool;
   //    nutRun36Ok : Bool;
   //    nutRun36NotOk : Bool;
   //    nutRun36Reserve : Bool;
   //    nutRun36TorqueHigh : Bool;
   //    nutRun36TorqueLow : Bool;
   //    nutRun36AngleHigh : Bool;
   //    nutRun36AngleLow : Bool;
   //    nutRun37NotMachined : Bool;
   //    nutRun37Ok : Bool;
   //    nutRun37NotOk : Bool;
   //    nutRun37Reserve : Bool;
   //    nutRun37TorqueHigh : Bool;
   //    nutRun37TorqueLow : Bool;
   //    nutRun37AngleHigh : Bool;
   //    nutRun37AngleLow : Bool;
   //    nutRun38NotMachined : Bool;
   //    nutRun38Ok : Bool;
   //    nutRun38NotOk : Bool;
   //    nutRun38Reserve : Bool;
   //    nutRun38TorqueHigh : Bool;
   //    nutRun38TorqueLow : Bool;
   //    nutRun38AngleHigh : Bool;
   //    nutRun38AngleLow : Bool;
   //    nutRun39NotMachined : Bool;
   //    nutRun39Ok : Bool;
   //    nutRun39NotOk : Bool;
   //    nutRun39Reserve : Bool;
   //    nutRun39TorqueHigh : Bool;
   //    nutRun39TorqueLow : Bool;
   //    nutRun39AngleHigh : Bool;
   //    nutRun39AngleLow : Bool;
   //    nutRun40NotMachined : Bool;
   //    nutRun40Ok : Bool;
   //    nutRun40NotOk : Bool;
   //    nutRun40Reserve : Bool;
   //    nutRun40TorqueHigh : Bool;
   //    nutRun40TorqueLow : Bool;
   //    nutRun40AngleHigh : Bool;
   //    nutRun40AngleLow : Bool;
   //    nutRun1Selected : Bool;
   //    nutRun2Selected : Bool;
   //    nutRun3Selected : Bool;
   //    nutRun4Selected : Bool;
   //    nutRun5Selected : Bool;
   //    nutRun6Selected : Bool;
   //    nutRun7Selected : Bool;
   //    nutRun8Selected : Bool;
   //    nutRun9Selected : Bool;
   //    nutRun10Selected : Bool;
   //    nutRun11Selected : Bool;
   //    nutRun12Selected : Bool;
   //    nutRun13Selected : Bool;
   //    nutRun14Selected : Bool;
   //    nutRun15Selected : Bool;
   //    nutRun16Selected : Bool;
   //    nutRun17Selected : Bool;
   //    nutRun18Selected : Bool;
   //    nutRun19Selected : Bool;
   //    nutRun20Selected : Bool;
   //    nutRun21Selected : Bool;
   //    nutRun22Selected : Bool;
   //    nutRun23Selected : Bool;
   //    nutRun24Selected : Bool;
   //    nutRun25Selected : Bool;
   //    nutRun26Selected : Bool;
   //    nutRun27Selected : Bool;
   //    nutRun28Selected : Bool;
   //    nutRun29Selected : Bool;
   //    nutRun30Selected : Bool;
   //    nutRun31Selected : Bool;
   //    nutRun32Selected : Bool;
   //    nutRun33Selected : Bool;
   //    nutRun34Selected : Bool;
   //    nutRun35Selected : Bool;
   //    nutRun36Selected : Bool;
   //    nutRun37Selected : Bool;
   //    nutRun38Selected : Bool;
   //    nutRun39Selected : Bool;
   //    nutRun40Selected : Bool;
   //    operation1 : Byte;
   //    operation2 : Byte;
   //    operation3 : Byte;
   //    operation4 : Byte;
   //    operation5 : Byte;
   //    operatorHelpPaletteNo1 : Byte;
   //    operatorHelpPaletteNo2 : Byte;
   //    operatorHelpCode1 : Byte;
   //    operatorHelpCode2 : Byte;
   //    operatorHelpCode3 : Byte;
   //    operatorHelpCode4 : Byte;
   //    charCodeAsc1 : Byte;
   //    charCodeAsc2 : Byte;
   //    charCodeAsc3 : Byte;
   //    charCodeAsc4 : Byte;
   //    res1886 : Array[1866..1889] of Byte;
   //    dataMediumReadStartAddr : Word;
   //    dataMediumWriteAddr : Word;
   //    dataMediumRwdNo : Byte;
   //    dataMediumDataValid : Bool;
   //    dataMediumDataModified : Bool;
   //    "res 8950" : Bool;
   //    dataMediumWriteBit : Bool;
   //    dataMediumReadBit : Bool;
   //    res18955 : Bool;
   //    res18956 : Bool;
   //    res18957 : Bool;
   //    res18960 : Struct
   //       toolDataChange : Array[1..96] of Bool;
   //       res_1908 : Array[1908..1927] of Byte;
   //       toolPreAlarmReached : Array[1..96] of Bool;
   //       res_1940 : Array[1940..1959] of Byte;
   //       toolAlarmReached : Array[1..96] of Bool;
   //       res_1972 : Array[1972..1991] of Byte;
   //       toolExtendedAlarmReached : Array[1..96] of Bool;
   //       res_2004 : Array[2004..2023] of Byte;
   //       toolDisabled : Array[1..96] of Bool;
   //       res_2036 : Array[2036..2055] of Byte;
   //       toolSetExtendedAlarm : Array[1..96] of Bool;
   //       res_2068 : Array[2068..2687] of Byte;
   //    END_STRUCT;
   //    powerup1ExecutableLeft : Bool;
   //    powerup1ExecutableRight : Bool;
   //    powerup2ExecutableLeft : Bool;
   //    powerup2ExecutableRight : Bool;
   //    powerup3ExecutableLeft : Bool;
   //    powerup3ExecutableRight : Bool;
   //    powerup4ExecutableLeft : Bool;
   //    powerup4ExecutableRight { ExternalAccessible := 'False'; ExternalVisible := 'False'; ExternalWritable := 'False'} : Bool;
   //    powerup5ExecutableLeft : Bool;
   //    powerup5ExecutableRight : Bool;
   //    powerup6ExecutableLeft : Bool;
   //    powerup6ExecutableRight : Bool;
   //    powerup7ExecutableLeft : Bool;
   //    powerup7ExecutableRight : Bool;
   //    powerup8ExecutableLeft : Bool;
   //    powerup8ExecutableRight : Bool;
   //    powerup9ExecutableLeft : Bool;
   //    powerup9ExecutableRight : Bool;
   //    powerup10ExecutableLeft : Bool;
   //    powerup10ExecutableRight : Bool;
   //    powerup11ExecutableLeft : Bool;
   //    powerup11ExecutableRight : Bool;
   //    powerup12ExecutableLeft : Bool;
   //    powerup12ExecutableRight : Bool;
   //    powerup13ExecutableLeft : Bool;
   //    powerup13ExecutableRight : Bool;
   //    powerup14ExecutableLeft : Bool;
   //    powerup14ExecutableRight : Bool;
   //    powerup15ExecutableLeft : Bool;
   //    powerup15ExecutableRight : Bool;
   //    powerup16ExecutableLeft : Bool;
   //    powerup16ExecutableRight : Bool;
   //    powerup17ExecutableLeft : Bool;
   //    powerup17ExecutableRight : Bool;
   //    powerup18ExecutableLeft : Bool;
   //    powerup18ExecutableRight : Bool;
   //    powerup19ExecutableLeft : Bool;
   //    powerup19ExecutableRight : Bool;
   //    powerup20ExecutableLeft : Bool;
   //    powerup20ExecutableRight : Bool;
   //    powerup21ExecutableLeft : Bool;
   //    powerup21ExecutableRight : Bool;
   //    powerup22ExecutableLeft : Bool;
   //    powerup22ExecutableRight : Bool;
   //    powerup23ExecutableLeft : Bool;
   //    powerup23ExecutableRight : Bool;
   //    powerup24ExecutableLeft : Bool;
   //    powerup24ExecutableRight : Bool;
   //    powerup25ExecutableLeft : Bool;
   //    powerup25ExecutableRight : Bool;
   //    powerup26ExecutableLeft : Bool;
   //    powerup26ExecutableRight : Bool;
   //    powerup27ExecutableLeft : Bool;
   //    powerup27ExecutableRight : Bool;
   //    powerup28ExecutableLeft : Bool;
   //    powerup28ExecutableRight : Bool;
   //    powerup29ExecutableLeft : Bool;
   //    powerup29ExecutableRight : Bool;
   //    powerup30ExecutableLeft : Bool;
   //    powerup30ExecutableRight : Bool;
   //    powerup31ExecutableLeft : Bool;
   //    powerup31ExecutableRight : Bool;
   //    powerup32ExecutableLeft : Bool;
   //    powerup32ExecutableRight : Bool;
   //    powerup33ExecutableLeft : Bool;
   //    powerup33ExecutableRight : Bool;
   //    powerup34ExecutableLeft : Bool;
   //    powerup34ExecutableRight : Bool;
   //    powerup35ExecutableLeft : Bool;
   //    powerup35ExecutableRight : Bool;
   //    powerup36ExecutableLeft : Bool;
   //    powerup36ExecutableRight : Bool;
   //    powerup37ExecutableLeft : Bool;
   //    powerup37ExecutableRight : Bool;
   //    powerup38ExecutableLeft : Bool;
   //    powerup38ExecutableRight : Bool;
   //    powerup39ExecutableLeft : Bool;
   //    powerup39ExecutableRight : Bool;
   //    powerup40ExecutableLeft : Bool;
   //    powerup40ExecutableRight : Bool;
   //    powerup41ExecutableLeft : Bool;
   //    powerup41ExecutableRight : Bool;
   //    powerup42ExecutableLeft : Bool;
   //    powerup42ExecutableRight : Bool;
   //    powerup43ExecutableLeft : Bool;
   //    powerup43ExecutableRight : Bool;
   //    powerup44ExecutableLeft : Bool;
   //    powerup44ExecutableRight : Bool;
   //    powerup45ExecutableLeft : Bool;
   //    powerup45ExecutableRight : Bool;
   //    powerup46ExecutableLeft : Bool;
   //    powerup46ExecutableRight : Bool;
   //    powerup47ExecutableLeft : Bool;
   //    powerup47ExecutableRight : Bool;
   //    powerup48ExecutableLeft : Bool;
   //    powerup48ExecutableRight : Bool;
   //    prealarmOnUnit1 : Bool;
   //    messageOnUnit1 : Bool;
   //    faSetupModeUnit1 : Bool;
   //    faSingleStepModeUnit1 : Bool;
   //    faSingleModeUnit1 : Bool;
   //    fctBit1ClampingUnit1 : Bool;
   //    fctBit2ClampingUnit1 : Bool;
   //    fctBit3ClampingUnit1 : Bool;
   //    prealarmOnUnit2 : Bool;
   //    messageOnUnit2 : Bool;
   //    faSetupModeUnit2 : Bool;
   //    faSingleStepModeUnit2 : Bool;
   //    faSingleModeUnit2 : Bool;
   //    fctBit1ClampingUnit2 : Bool;
   //    fctBit2ClampingUnit2 : Bool;
   //    fctBit3ClampingUnit2 : Bool;
   //    prealarmOnUnit3 : Bool;
   //    messageOnUnit3 : Bool;
   //    faSetupModeUnit3 : Bool;
   //    faSingleStepModeUnit3 : Bool;
   //    faSingleModeUnit3 : Bool;
   //    fctBit1ClampingUnit3 : Bool;
   //    fctBit2ClampingUnit3 : Bool;
   //    fctBit3ClampingUnit3 : Bool;
   //    prealarmOnUnit4 : Bool;
   //    messageOnUnit4 : Bool;
   //    faSetupModeUnit4 : Bool;
   //    faSingleStepModeUnit4 : Bool;
   //    faSingleModeUnit4 : Bool;
   //    fctBit1ClampingUnit4 : Bool;
   //    fctBit2ClampingUnit4 : Bool;
   //    fctBit3ClampingUnit4 : Bool;
   //    prealarmOnUnit5 : Bool;
   //    messageOnUnit5 : Bool;
   //    faSetupModeUnit5 : Bool;
   //    faSingleStepModeUnit5 : Bool;
   //    faSingleModeUnit5 : Bool;
   //    fctBit1ClampingUnit5 : Bool;
   //    fctBit2ClampingUnit5 : Bool;
   //    fctBit3ClampingUnit5 : Bool;
   //    prealarmOnUnit6 : Bool;
   //    messageOnUnit6 : Bool;
   //    faSetupModeUnit6 : Bool;
   //    faSingleStepModeUnit6 : Bool;
   //    faSingleModeUnit6 : Bool;
   //    fctBit1ClampingUnit6 : Bool;
   //    fctBit2ClampingUnit6 : Bool;
   //    fctBit3ClampingUnit6 : Bool;
   //    prealarmOnUnit7 : Bool;
   //    messageOnUnit7 : Bool;
   //    faSetupModeUnit7 : Bool;
   //    faSingleStepModeUnit7 : Bool;
   //    faSingleModeUnit7 : Bool;
   //    fctBit1ClampingUnit7 : Bool;
   //    fctBit2ClampingUnit7 : Bool;
   //    fctBit3ClampingUnit7 : Bool;
   //    prealarmOnUnit8 : Bool;
   //    messageOnUnit8 : Bool;
   //    faSetupModeUnit8 : Bool;
   //    faSingleStepModeUnit8 : Bool;
   //    faSingleModeUnit8 : Bool;
   //    fctBit1ClampingUnit8 : Bool;
   //    fctBit2ClampingUnit8 : Bool;
   //    fctBit3ClampingUnit8 : Bool;
   //    prealarmOnUnit9 : Bool;
   //    messageOnUnit9 : Bool;
   //    faSetupModeUnit9 : Bool;
   //    faSingleStepModeUnit9 : Bool;
   //    faSingleModeUnit9 : Bool;
   //    fctBit1ClampingUnit9 : Bool;
   //    fctBit2ClampingUnit9 : Bool;
   //    fctBit3ClampingUnit9 : Bool;
   //    prealarmOnUnit10 : Bool;
   //    messageOnUnit10 : Bool;
   //    faSetupModeUnit10 : Bool;
   //    faSingleStepModeUnit10 : Bool;
   //    faSingleModeUnit10 : Bool;
   //    fctBit1ClampingUnit10 : Bool;
   //    fctBit2ClampingUnit10 : Bool;
   //    fctBit3ClampingUnit10 : Bool;
   //    prealarmOnUnit11 : Bool;
   //    messageOnUnit11 : Bool;
   //    faSetupModeUnit11 : Bool;
   //    faSingleStepModeUnit11 : Bool;
   //    faSingleModeUnit11 : Bool;
   //    fctBit1ClampingUnit11 : Bool;
   //    fctBit2ClampingUnit11 : Bool;
   //    fctBit3ClampingUnit11 : Bool;
   //    prealarmOnUnit12 : Bool;
   //    messageOnUnit12 : Bool;
   //    faSetupModeUnit12 : Bool;
   //    faSingleStepModeUnit12 : Bool;
   //    faSingleModeUnit12 : Bool;
   //    fctBit1ClampingUnit12 : Bool;
   //    fctBit2ClampingUnit12 : Bool;
   //    fctBit3ClampingUnit12 : Bool;
   //    prealarmOnUnit13 : Bool;
   //    messageOnUnit13 : Bool;
   //    faSetupModeUnit13 : Bool;
   //    faSingleStepModeUnit13 : Bool;
   //    faSingleModeUnit13 : Bool;
   //    fctBit1ClampingUnit13 : Bool;
   //    fctBit2ClampingUnit13 : Bool;
   //    fctBit3ClampingUnit13 : Bool;
   //    prealarmOnUnit14 : Bool;
   //    messageOnUnit14 : Bool;
   //    faSetupModeUnit14 : Bool;
   //    faSingleStepModeUnit14 : Bool;
   //    faSingleModeUnit14 : Bool;
   //    fctBit1ClampingUnit14 : Bool;
   //    fctBit2ClampingUnit14 : Bool;
   //    fctBit3ClampingUnit14 : Bool;
   //    prealarmOnUnit15 : Bool;
   //    messageOnUnit15 : Bool;
   //    faSetupModeUnit15 : Bool;
   //    faSingleStepModeUnit15 : Bool;
   //    faSingleModeUnit15 : Bool;
   //    fctBit1ClampingUnit15 : Bool;
   //    fctBit2ClampingUnit15 : Bool;
   //    fctBit3ClampingUnit15 : Bool;
   //    prealarmOnUnit16 : Bool;
   //    messageOnUnit16 : Bool;
   //    faSetupModeUnit16 : Bool;
   //    faSingleStepModeUnit16 : Bool;
   //    faSingleModeUnit16 : Bool;
   //    fctBit1ClampingUnit16 : Bool;
   //    fctBit2ClampingUnit16 : Bool;
   //    fctBit3ClampingUnit16 : Bool;
   //    prealarmOnUnit17 : Bool;
   //    messageOnUnit17 : Bool;
   //    faSetupModeUnit17 : Bool;
   //    faSingleStepModeUnit17 : Bool;
   //    faSingleModeUnit17 : Bool;
   //    fctBit1ClampingUnit17 : Bool;
   //    fctBit2ClampingUnit17 : Bool;
   //    fctBit3ClampingUnit17 : Bool;
   //    prealarmOnUnit18 : Bool;
   //    messageOnUnit18 : Bool;
   //    faSetupModeUnit18 : Bool;
   //    faSingleStepModeUnit18 : Bool;
   //    faSingleModeUnit18 : Bool;
   //    fctBit1ClampingUnit18 : Bool;
   //    fctBit2ClampingUnit18 : Bool;
   //    fctBit3ClampingUnit18 : Bool;
   //    prealarmOnUnit19 : Bool;
   //    messageOnUnit19 : Bool;
   //    faSetupModeUnit19 : Bool;
   //    faSingleStepModeUnit19 : Bool;
   //    faSingleModeUnit19 : Bool;
   //    fctBit1ClampingUnit19 : Bool;
   //    fctBit2ClampingUnit19 : Bool;
   //    fctBit3ClampingUnit19 : Bool;
   //    prealarmOnUnit20 : Bool;
   //    messageOnUnit20 : Bool;
   //    faSetupModeUnit20 : Bool;
   //    faSingleStepModeUnit20 : Bool;
   //    faSingleModeUnit20 : Bool;
   //    fctBit1ClampingUnit20 : Bool;
   //    fctBit2ClampingUnit20 : Bool;
   //    fctBit3ClampingUnit20 : Bool;
   //    prealarmOnUnit21 : Bool;
   //    messageOnUnit21 : Bool;
   //    faSetupModeUnit21 : Bool;
   //    faSingleStepModeUnit21 : Bool;
   //    faSingleModeUnit21 : Bool;
   //    fctBit1ClampingUnit21 : Bool;
   //    fctBit2ClampingUnit21 : Bool;
   //    fctBit3ClampingUnit21 : Bool;
   //    prealarmOnUnit22 : Bool;
   //    messageOnUnit22 : Bool;
   //    faSetupModeUnit22 : Bool;
